DATA_BLOCK "BM_GRW_REC_BOOL"   // DB701
{ S7_Optimized_Access := 'FALSE' }
VERSION : 0.0
// --------------------------------------------------------------------------------
// program:             GRW_REC_BOOL
// description :        bool data for growth record
// name:                mb
// date        :        27.11.09 
// --------------------------------------------------------------------------------
   VAR
      phase_restart : Bool;   // Phase wurde neu gestartet
      phase_spare_02 : Bool;
      phase_spare_03 : Bool;
      phase_spare_04 : Bool;
      phase_spare_05 : Bool;
      phase_spare_06 : Bool;
      phase_spare_07 : Bool;
      phase_spare_08 : Bool;
      phase_spare_09 : Bool;
      phase_spare_10 : Bool;   // pump down
      pd_min_prs_reached : Bool;   // min. Druck erreicht
      pd_failed : Bool;   // Leckrate (0=ok/1=nicht ok)
      pd_new_seed : Bool;   // neuer Impfling bei Prozesstart
      pd_spare_04 : Bool;
      pd_spare_05 : Bool;
      pd_spare_06 : Bool;
      pd_spare_07 : Bool;
      pd_spare_08 : Bool;
      pd_spare_09 : Bool;
      pd_spare_10 : Bool;   // melting
      me_completed : Bool;   // Einschmelzen beendet (von Kamera erkannt)
      me_spare_02 : Bool;
      me_spare_03 : Bool;
      me_spare_04 : Bool;
      me_spare_05 : Bool;
      me_spare_06 : Bool;
      me_spare_07 : Bool;
      me_spare_08 : Bool;
      me_spare_09 : Bool;
      me_spare_10 : Bool;   // dipping
      di_new_seed : Bool;   // alter oder neuer Impfling (0=alt/1=neu)
      di_shield_dn : Bool;   // Trichter ist unten
      di_spare_03 : Bool;
      di_spare_04 : Bool;
      di_spare_05 : Bool;
      di_spare_06 : Bool;
      di_spare_07 : Bool;
      di_spare_08 : Bool;
      di_spare_09 : Bool;
      di_spare_10 : Bool;   // neck
      ne_spare_01 : Bool;
      ne_spare_02 : Bool;
      ne_spare_03 : Bool;
      ne_spare_04 : Bool;
      ne_spare_05 : Bool;
      ne_spare_06 : Bool;
      ne_spare_07 : Bool;
      ne_spare_08 : Bool;
      ne_spare_09 : Bool;
      ne_spare_10 : Bool;   // shoulder
      sh_spare_01 : Bool;
      sh_spare_02 : Bool;
      sh_spare_03 : Bool;
      sh_spare_04 : Bool;
      sh_spare_05 : Bool;
      sh_spare_06 : Bool;
      sh_spare_07 : Bool;
      sh_spare_08 : Bool;
      sh_spare_09 : Bool;
      sh_spare_10 : Bool;   // body
      by_spare_01 : Bool;
      by_spare_02 : Bool;
      by_spare_03 : Bool;
      by_spare_04 : Bool;
      by_spare_05 : Bool;
      by_spare_06 : Bool;
      by_spare_07 : Bool;
      by_spare_08 : Bool;
      by_spare_09 : Bool;
      by_spare_10 : Bool;   // endcone
      ec_spare_01 : Bool;
      ec_spare_02 : Bool;
      ec_spare_03 : Bool;
      ec_spare_04 : Bool;
      ec_spare_05 : Bool;
      ec_spare_06 : Bool;
      ec_spare_07 : Bool;
      ec_spare_08 : Bool;
      ec_spare_09 : Bool;
      ec_spare_10 : Bool;   // shut down
      sd_spare_01 : Bool;
      sd_spare_02 : Bool;
      sd_spare_03 : Bool;
      sd_spare_04 : Bool;
      sd_spare_05 : Bool;
      sd_spare_06 : Bool;
      sd_spare_07 : Bool;
      sd_spare_08 : Bool;
      sd_spare_09 : Bool;
      sd_spare_10 : Bool;   // removal
      re_active : Bool;   // Entnahme wurde ausgef黨rt
      re_spare_02 : Bool;
      re_spare_03 : Bool;
      re_spare_04 : Bool;
      re_spare_05 : Bool;
      re_spare_06 : Bool;
      re_spare_07 : Bool;
      re_spare_08 : Bool;
      re_spare_09 : Bool;
      re_spare_10 : Bool;   // melting back
      mb_spare_01 : Bool;
      mb_spare_02 : Bool;
      mb_spare_03 : Bool;
      mb_spare_04 : Bool;
      mb_spare_05 : Bool;
      mb_spare_06 : Bool;
      mb_spare_07 : Bool;
      mb_spare_08 : Bool;
      mb_spare_09 : Bool;
      mb_spare_10 : Bool;   // interne Speicherbits
      pd_sps_spare_01 : Bool;
      pd_sps_spare_02 : Bool;
      pd_sps_spare_03 : Bool;
      pd_sps_spare_04 : Bool;
      pd_sps_spare_05 : Bool;
      pd_sps_spare_06 : Bool;
      pd_sps_spare_07 : Bool;
      pd_sps_spare_08 : Bool;
      pd_sps_spare_09 : Bool;
      pd_sps_spare_10 : Bool;
      me_sps_spare_01 : Bool;
      me_sps_spare_02 : Bool;
      me_sps_spare_03 : Bool;
      me_sps_spare_04 : Bool;
      me_sps_spare_05 : Bool;
      me_sps_spare_06 : Bool;
      me_sps_spare_07 : Bool;
      me_sps_spare_08 : Bool;
      me_sps_spare_09 : Bool;
      me_sps_spare_10 : Bool;
      di_init_melt_temp : Bool;   // speichern Anfangs-Schmelzbadtemp. ausgef黨rt
      di_time_until_dip : Bool;   // speichern der Zeit bis Impfling in Schmelze ausgef黨rt
      di_sps_spare_03 : Bool;
      di_sps_spare_04 : Bool;
      di_sps_spare_05 : Bool;
      di_sps_spare_06 : Bool;
      di_sps_spare_07 : Bool;
      di_sps_spare_08 : Bool;
      di_sps_spare_09 : Bool;
      di_sps_spare_10 : Bool;
      ne_init_xt_pos : Bool;   // speichern Anfangs-Kristallpos. ausgef黨rt
      ne_init_cr_pos : Bool;   // speichern Anfangs-Tiegelposition ausgef黨rt
      ne_init_melt_temp : Bool;   // speichern Anfangs-Schmelzbadtemp. ausgef黨rt
      ne_low_temp_inc : Bool;   // speichern niedrigstes Temp.Inkrement ausgef黨rt
      ne_init_htr_temp : Bool;   // speichern Heizertemp
      ne_sps_spare_06 : Bool;
      ne_sps_spare_07 : Bool;
      ne_sps_spare_08 : Bool;
      ne_sps_spare_09 : Bool;
      ne_sps_spare_10 : Bool;
      sh_start_dia : Bool;   // speichern Startdurchmesser ausgef黨rt
      sh_init_htr_temp : Bool;   // speichern Heizertemp
      sh_sps_spare_03 : Bool;
      sh_sps_spare_04 : Bool;
      sh_sps_spare_05 : Bool;
      sh_sps_spare_06 : Bool;
      sh_sps_spare_07 : Bool;
      sh_sps_spare_08 : Bool;
      sh_sps_spare_09 : Bool;
      sh_sps_spare_10 : Bool;
      by_low_temp_inc : Bool;   // speichern niedrigstes Temp.Inkrement ausgef黨rt
      by_first_dia : Bool;   // speichern Startdurchmesser ausgef黨rt
      by_init_htr_temp : Bool;   // speichern Heizertemp
      by_sps_spare_04 : Bool;
      by_sps_spare_05 : Bool;
      by_sps_spare_06 : Bool;
      by_sps_spare_07 : Bool;
      by_sps_spare_08 : Bool;
      by_sps_spare_09 : Bool;
      by_sps_spare_10 : Bool;
      ec_init_htr_temp : Bool;   // speichern Heizertemp
      ec_sps_spare_02 : Bool;
      ec_sps_spare_03 : Bool;
      ec_sps_spare_04 : Bool;
      ec_sps_spare_05 : Bool;
      ec_sps_spare_06 : Bool;
      ec_sps_spare_07 : Bool;
      ec_sps_spare_08 : Bool;
      ec_sps_spare_09 : Bool;
      ec_sps_spare_10 : Bool;
      sd_sps_spare_01 : Bool;
      sd_sps_spare_02 : Bool;
      sd_sps_spare_03 : Bool;
      sd_sps_spare_04 : Bool;
      sd_sps_spare_05 : Bool;
      sd_sps_spare_06 : Bool;
      sd_sps_spare_07 : Bool;
      sd_sps_spare_08 : Bool;
      sd_sps_spare_09 : Bool;
      sd_sps_spare_10 : Bool;
      re_next_cr_pos : Bool;   // speichern Tiegelposition f黵 n鋍hstes Ankeimen ausgef黨rt
      re_sps_spare_02 : Bool;
      re_sps_spare_03 : Bool;
      re_sps_spare_04 : Bool;
      re_sps_spare_05 : Bool;
      re_sps_spare_06 : Bool;
      re_sps_spare_07 : Bool;
      re_sps_spare_08 : Bool;
      re_sps_spare_09 : Bool;
      re_sps_spare_10 : Bool;
      mb_sps_spare_01 : Bool;
      mb_sps_spare_02 : Bool;
      mb_sps_spare_03 : Bool;
      mb_sps_spare_04 : Bool;
      mb_sps_spare_05 : Bool;
      mb_sps_spare_06 : Bool;
      mb_sps_spare_07 : Bool;
      mb_sps_spare_08 : Bool;
      mb_sps_spare_09 : Bool;
      mb_sps_spare_10 : Bool;
   END_VAR
BEGIN
END_DATA_BLOCK

DATA_BLOCK "BM_GRW_REC_DINT"   // DB702
{ S7_Optimized_Access := 'FALSE' }
VERSION : 0.0
// --------------------------------------------------------------------------------
// program     :        GRW_REC_DINT
// description :        dint data for growth record
// name        :        mb
// date        :        27.11.09
// --------------------------------------------------------------------------------
   VAR
      elapsed_time : DInt;   // gesamte Prozesszeit
      phase_spare_02 : DInt;
      phase_spare_03 : DInt;
      phase_spare_04 : DInt;
      phase_spare_05 : DInt;
      phase_spare_06 : DInt;
      phase_spare_07 : DInt;
      phase_spare_08 : DInt;
      phase_spare_09 : DInt;
      phase_spare_10 : DInt;
      pd_elapsed_time : DInt;   // insgesamt vergangene Prozesszeit
      pd_phase_time : DInt;   // aktuelle/letzte Phasendauer
      pd_to_min_prs : DInt;   // Zeit bis Enddruck erreicht
      pd_retry : DInt;
      pd_spare_05 : DInt;
      pd_spare_06 : DInt;
      pd_spare_07 : DInt;
      pd_spare_08 : DInt;
      pd_spare_09 : DInt;
      pd_spare_10 : DInt;
      me_elapsed_time : DInt;   // insgesamt vergangene Prozesszeit
      me_phase_time : DInt;   // aktuelle/letzte Phasendauer
      me_melt_time : DInt;   // Zeit bis Aufschmelzen beendet
      me_spare_04 : DInt;
      me_spare_05 : DInt;
      me_spare_06 : DInt;
      me_spare_07 : DInt;
      me_spare_08 : DInt;
      me_spare_09 : DInt;
      me_spare_10 : DInt;
      di_elapsed_time : DInt;   // insgesamt vergangene Prozesszeit
      di_phase_time : DInt;   // aktuelle/letzte Phasendauer
      di_shield_dn : DInt;   // Zeit bis Trichter unten
      di_time_until_dip : DInt;   // Zeit bis Impfling in Schmelze
      di_spare_05 : DInt;
      di_spare_06 : DInt;
      di_spare_07 : DInt;
      di_spare_08 : DInt;
      di_spare_09 : DInt;
      di_spare_10 : DInt;
      ne_elapsed_time : DInt;   // insgesamt vergangene Prozesszeit
      ne_phase_time : DInt;   // aktuelle/letzte Phasendauer
      ne_spare_03 : DInt;
      ne_spare_04 : DInt;
      ne_spare_05 : DInt;
      ne_spare_06 : DInt;
      ne_spare_07 : DInt;
      ne_spare_08 : DInt;
      ne_spare_09 : DInt;
      ne_spare_10 : DInt;
      sh_elapsed_time : DInt;   // insgesamt vergangene Prozesszeit
      sh_phase_time : DInt;   // aktuelle/letzte Phasendauer
      sh_spare_03 : DInt;
      sh_spare_04 : DInt;
      sh_spare_05 : DInt;
      sh_spare_06 : DInt;
      sh_spare_07 : DInt;
      sh_spare_08 : DInt;
      sh_spare_09 : DInt;
      sh_spare_10 : DInt;
      by_elapsed_time : DInt;   // insgesamt vergangene Prozesszeit
      by_phase_time : DInt;   // aktuelle/letzte Phasendauer
      by_spare_03 : DInt;
      by_spare_04 : DInt;
      by_spare_05 : DInt;
      by_spare_06 : DInt;
      by_spare_07 : DInt;
      by_spare_08 : DInt;
      by_spare_09 : DInt;
      by_spare_10 : DInt;
      ec_elapsed_time : DInt;   // insgesamt vergangene Prozesszeit
      ec_phase_time : DInt;   // aktuelle/letzte Phasendauer
      ec_spare_03 : DInt;
      ec_spare_04 : DInt;
      ec_spare_05 : DInt;
      ec_spare_06 : DInt;
      ec_spare_07 : DInt;
      ec_spare_08 : DInt;
      ec_spare_09 : DInt;
      ec_spare_10 : DInt;
      sd_elapsed_time : DInt;   // insgesamt vergangene Prozesszeit
      sd_phase_time : DInt;   // aktuelle/letzte Phasendauer
      sd_spare_03 : DInt;
      sd_spare_04 : DInt;
      sd_spare_05 : DInt;
      sd_spare_06 : DInt;
      sd_spare_07 : DInt;
      sd_spare_08 : DInt;
      sd_spare_09 : DInt;
      sd_spare_10 : DInt;
      re_elapsed_time : DInt;   // insgesamt vergangene Prozesszeit
      re_phase_time : DInt;   // aktuelle/letzte Phasendauer
      re_spare_03 : DInt;
      re_spare_04 : DInt;
      re_spare_05 : DInt;
      re_spare_06 : DInt;
      re_spare_07 : DInt;
      re_spare_08 : DInt;
      re_spare_09 : DInt;
      re_spare_10 : DInt;
      mb_elapsed_time : DInt;   // insgesamt vergangene Prozesszeit
      mb_phase_time : DInt;   // aktuelle/letzte Phasendauer
      mb_spare_03 : DInt;
      mb_spare_04 : DInt;
      mb_spare_05 : DInt;
      mb_spare_06 : DInt;
      mb_spare_07 : DInt;
      mb_spare_08 : DInt;
      mb_spare_09 : DInt;
      mb_spare_10 : DInt;
   END_VAR
BEGIN
END_DATA_BLOCK

DATA_BLOCK "BM_GRW_REC_REAL"   // DB703
{ S7_Optimized_Access := 'FALSE' }
VERSION : 0.0
// --------------------------------------------------------------------------------
// program:             GRW_REC_REAL
// description :        REAL data for growth record
// name:                mb
// date        :        23.11.09
// --------------------------------------------------------------------------------
   VAR
      htr_pwr_csp : Real;   // heater power consumption
      ar_gas_csp : Real;   // argon gas consumption
      phase_spare_03 : Real;
      phase_spare_04 : Real;
      phase_spare_05 : Real;
      phase_spare_06 : Real;
      phase_spare_07 : Real;
      phase_spare_08 : Real;
      phase_spare_09 : Real;
      phase_spare_10 : Real;
      phase_spare_11 : Real;
      phase_spare_12 : Real;
      phase_spare_13 : Real;
      phase_spare_14 : Real;
      phase_spare_15 : Real;
      phase_spare_16 : Real;
      phase_spare_17 : Real;
      phase_spare_18 : Real;
      phase_spare_19 : Real;
      phase_spare_20 : Real;
      phase_spare_21 : Real;
      phase_spare_22 : Real;
      phase_spare_23 : Real;
      phase_spare_24 : Real;
      phase_spare_25 : Real;
      phase_spare_26 : Real;
      phase_spare_27 : Real;
      phase_spare_28 : Real;
      phase_spare_29 : Real;
      phase_spare_30 : Real;
      phase_spare_31 : Real;
      phase_spare_32 : Real;
      phase_spare_33 : Real;
      phase_spare_34 : Real;
      phase_spare_35 : Real;
      phase_spare_36 : Real;
      phase_spare_37 : Real;
      phase_spare_38 : Real;
      phase_spare_39 : Real;
      phase_spare_40 : Real;
      pd_final_prs : Real;   // erreichter Enddruck
      pd_leakrate : Real;   // Leckrate
      pd_spare_03 : Real;
      pd_spare_04 : Real;
      pd_spare_05 : Real;
      pd_spare_06 : Real;
      pd_spare_07 : Real;
      pd_spare_08 : Real;
      pd_spare_09 : Real;
      pd_spare_10 : Real;
      pd_spare_11 : Real;
      pd_spare_12 : Real;
      pd_spare_13 : Real;
      pd_spare_14 : Real;
      pd_spare_15 : Real;
      pd_spare_16 : Real;
      pd_spare_17 : Real;
      pd_spare_18 : Real;
      pd_spare_19 : Real;
      pd_spare_20 : Real;
      pd_spare_21 : Real;
      pd_spare_22 : Real;
      pd_spare_23 : Real;
      pd_spare_24 : Real;
      pd_spare_25 : Real;
      pd_spare_26 : Real;
      pd_spare_27 : Real;
      pd_spare_28 : Real;
      pd_spare_29 : Real;
      pd_spare_30 : Real;
      pd_spare_31 : Real;
      pd_spare_32 : Real;
      pd_spare_33 : Real;
      pd_spare_34 : Real;
      pd_spare_35 : Real;
      pd_spare_36 : Real;
      pd_spare_37 : Real;
      pd_spare_38 : Real;
      pd_spare_39 : Real;
      pd_spare_40 : Real;
      me_spare_01 : Real;
      me_spare_02 : Real;
      me_spare_03 : Real;
      me_spare_04 : Real;
      me_spare_05 : Real;
      me_spare_06 : Real;
      me_spare_07 : Real;
      me_spare_08 : Real;
      me_spare_09 : Real;
      me_spare_10 : Real;
      me_spare_11 : Real;
      me_spare_12 : Real;
      me_spare_13 : Real;
      me_spare_14 : Real;
      me_spare_15 : Real;
      me_spare_16 : Real;
      me_spare_17 : Real;
      me_spare_18 : Real;
      me_spare_19 : Real;
      me_spare_20 : Real;
      me_spare_21 : Real;
      me_spare_22 : Real;
      me_spare_23 : Real;
      me_spare_24 : Real;
      me_spare_25 : Real;
      me_spare_26 : Real;
      me_spare_27 : Real;
      me_spare_28 : Real;
      me_spare_29 : Real;
      me_spare_30 : Real;
      me_spare_31 : Real;
      me_spare_32 : Real;
      me_spare_33 : Real;
      me_spare_34 : Real;
      me_spare_35 : Real;
      me_spare_36 : Real;
      me_spare_37 : Real;
      me_spare_38 : Real;
      me_spare_39 : Real;
      me_spare_40 : Real;
      di_init_melt_temp : Real;   // Anfangs-Schmelzbadtemp.
      di_final_htr_1_pwr : Real;   // Heizer 1 Leistung am Phasenende
      di_spare_03 : Real;
      di_spare_04 : Real;
      di_spare_05 : Real;
      di_spare_06 : Real;
      di_spare_07 : Real;
      di_spare_08 : Real;
      di_spare_09 : Real;
      di_spare_10 : Real;
      di_spare_11 : Real;
      di_spare_12 : Real;
      di_spare_13 : Real;
      di_spare_14 : Real;
      di_spare_15 : Real;
      di_spare_16 : Real;
      di_spare_17 : Real;
      di_spare_18 : Real;
      di_spare_19 : Real;
      di_spare_20 : Real;
      di_spare_21 : Real;
      di_spare_22 : Real;
      di_spare_23 : Real;
      di_spare_24 : Real;
      di_spare_25 : Real;
      di_spare_26 : Real;
      di_spare_27 : Real;
      di_spare_28 : Real;
      di_spare_29 : Real;
      di_spare_30 : Real;
      di_spare_31 : Real;
      di_spare_32 : Real;
      di_spare_33 : Real;
      di_spare_34 : Real;
      di_spare_35 : Real;
      di_spare_36 : Real;
      di_spare_37 : Real;
      di_spare_38 : Real;
      di_spare_39 : Real;
      di_spare_40 : Real;
      ne_init_cr_pos : Real;   // Anfangs-Tiegelpos.
      ne_init_melt_temp : Real;   // Anfangs-Schmelzbadtemp.
      ne_final_melt_temp : Real;   // finale-Schmelzbadtemp.
      ne_low_temp_inc : Real;   // niedrigstes Temp.Inc.
      ne_final_temp_inc : Real;   // finales Temp.Inc.
      ne_phase_avg_spd : Real;   // Durchschnittl. Ziehgeschwindigkeit (gesamte Halsl鋘ge)
      ne_final_avg_spd : Real;   // finale Durchschnittl. Ziehgeschwindigkeit
      ne_final_htr_1_pwr : Real;   // Heizer 1 Leistung am Phasenende
      ne_spare_09 : Real;
      ne_spare_10 : Real;
      ne_spare_11 : Real;
      ne_spare_12 : Real;
      ne_spare_13 : Real;
      ne_spare_14 : Real;
      ne_spare_15 : Real;
      ne_spare_16 : Real;
      ne_spare_17 : Real;
      ne_spare_18 : Real;
      ne_spare_19 : Real;
      ne_spare_20 : Real;
      ne_spare_21 : Real;
      ne_spare_22 : Real;
      ne_spare_23 : Real;
      ne_spare_24 : Real;
      ne_spare_25 : Real;
      ne_spare_26 : Real;
      ne_spare_27 : Real;
      ne_spare_28 : Real;
      ne_spare_29 : Real;
      ne_spare_30 : Real;
      ne_spare_31 : Real;
      ne_spare_32 : Real;
      ne_spare_33 : Real;
      ne_spare_34 : Real;
      ne_spare_35 : Real;
      ne_spare_36 : Real;
      ne_spare_37 : Real;
      ne_spare_38 : Real;
      ne_spare_39 : Real;
      ne_spare_40 : Real;
      sh_phase_avg_grth : Real;   // Durchschnittl. Wachstumsgeschwindigkeit (gesamte Schulter)
      sh_final_temp_inc : Real;   // finales Temp.Inc.
      sh_weight : Real;   // Gewicht der Schulter
      sh_final_htr_1_pwr : Real;   // Heizer 1 Leistung am Phasenende
      sh_spare_05 : Real;
      sh_spare_06 : Real;
      sh_spare_07 : Real;
      sh_spare_08 : Real;
      sh_spare_09 : Real;
      sh_spare_10 : Real;
      sh_spare_11 : Real;
      sh_spare_12 : Real;
      sh_spare_13 : Real;
      sh_spare_14 : Real;
      sh_spare_15 : Real;
      sh_spare_16 : Real;
      sh_spare_17 : Real;
      sh_spare_18 : Real;
      sh_spare_19 : Real;
      sh_spare_20 : Real;
      sh_spare_21 : Real;
      sh_spare_22 : Real;
      sh_spare_23 : Real;
      sh_spare_24 : Real;
      sh_spare_25 : Real;
      sh_spare_26 : Real;
      sh_spare_27 : Real;
      sh_spare_28 : Real;
      sh_spare_29 : Real;
      sh_spare_30 : Real;
      sh_spare_31 : Real;
      sh_spare_32 : Real;
      sh_spare_33 : Real;
      sh_spare_34 : Real;
      sh_spare_35 : Real;
      sh_spare_36 : Real;
      sh_spare_37 : Real;
      sh_spare_38 : Real;
      sh_spare_39 : Real;
      sh_spare_40 : Real;
      by_phase_avg_spd : Real;   // Durchschnittl. Ziehgeschwindigkeit (gesamt)
      by_final_avg_spd : Real;   // finale Durchschnittl. Ziehgeschwindigkeit
      by_low_temp_inc : Real;   // niedrigstes Temp.Inc.
      by_final_temp_inc : Real;   // finales Temp.Inc.
      by_avg_dia : Real;   // Durchschnittl. Durchmesser
      by_weight : Real;   // Gewicht vom Stab
      by_lenght : Real;   // Stabl鋘ge
      by_total_length : Real;   // Gesamtl鋘ge
      by_rem_cr_wgt : Real;   // verbleibende Siliziummenge im Tiegel
      by_final_cr_pos : Real;   // finale Tiegelpos.
      by_final_htr_1_pwr : Real;   // Heizer 1 Leistung am Phasenende
      by_spare_12 : Real;
      by_spare_13 : Real;
      by_spare_14 : Real;
      by_spare_15 : Real;
      by_spare_16 : Real;
      by_spare_17 : Real;
      by_spare_18 : Real;
      by_spare_19 : Real;
      by_spare_20 : Real;
      by_spare_21 : Real;
      by_spare_22 : Real;
      by_spare_23 : Real;
      by_spare_24 : Real;
      by_spare_25 : Real;
      by_spare_26 : Real;
      by_spare_27 : Real;
      by_spare_28 : Real;
      by_spare_29 : Real;
      by_spare_30 : Real;
      by_spare_31 : Real;
      by_spare_32 : Real;
      by_spare_33 : Real;
      by_spare_34 : Real;
      by_spare_35 : Real;
      by_spare_36 : Real;
      by_spare_37 : Real;
      by_spare_38 : Real;
      by_spare_39 : Real;
      by_spare_40 : Real;
      ec_phase_avg_spd : Real;   // Durchschnittl. Ziehgeschwindigkeit (gesamt)
      ec_final_temp_inc : Real;   // finales Temp.Inc.
      ec_weight : Real;   // Gewicht vom Endkonus
      ec_rem_cr_wgt : Real;   // verbleibende Siliziummenge im Tiegel
      ec_final_htr_1_pwr : Real;   // Heizer 1 Leistung am Phasenende
      ec_spare_06 : Real;
      ec_spare_07 : Real;
      ec_spare_08 : Real;
      ec_spare_09 : Real;
      ec_spare_10 : Real;
      ec_spare_11 : Real;
      ec_spare_12 : Real;
      ec_spare_13 : Real;
      ec_spare_14 : Real;
      ec_spare_15 : Real;
      ec_spare_16 : Real;
      ec_spare_17 : Real;
      ec_spare_18 : Real;
      ec_spare_19 : Real;
      ec_spare_20 : Real;
      ec_spare_21 : Real;
      ec_spare_22 : Real;
      ec_spare_23 : Real;
      ec_spare_24 : Real;
      ec_spare_25 : Real;
      ec_spare_26 : Real;
      ec_spare_27 : Real;
      ec_spare_28 : Real;
      ec_spare_29 : Real;
      ec_spare_30 : Real;
      ec_spare_31 : Real;
      ec_spare_32 : Real;
      ec_spare_33 : Real;
      ec_spare_34 : Real;
      ec_spare_35 : Real;
      ec_spare_36 : Real;
      ec_spare_37 : Real;
      ec_spare_38 : Real;
      ec_spare_39 : Real;
      ec_spare_40 : Real;
      sd_spare_01 : Real;
      sd_spare_02 : Real;
      sd_spare_03 : Real;
      sd_spare_04 : Real;
      sd_spare_05 : Real;
      sd_spare_06 : Real;
      sd_spare_07 : Real;
      sd_spare_08 : Real;
      sd_spare_09 : Real;
      sd_spare_10 : Real;
      sd_spare_11 : Real;
      sd_spare_12 : Real;
      sd_spare_13 : Real;
      sd_spare_14 : Real;
      sd_spare_15 : Real;
      sd_spare_16 : Real;
      sd_spare_17 : Real;
      sd_spare_18 : Real;
      sd_spare_19 : Real;
      sd_spare_20 : Real;
      sd_spare_21 : Real;
      sd_spare_22 : Real;
      sd_spare_23 : Real;
      sd_spare_24 : Real;
      sd_spare_25 : Real;
      sd_spare_26 : Real;
      sd_spare_27 : Real;
      sd_spare_28 : Real;
      sd_spare_29 : Real;
      sd_spare_30 : Real;
      sd_spare_31 : Real;
      sd_spare_32 : Real;
      sd_spare_33 : Real;
      sd_spare_34 : Real;
      sd_spare_35 : Real;
      sd_spare_36 : Real;
      sd_spare_37 : Real;
      sd_spare_38 : Real;
      sd_spare_39 : Real;
      sd_spare_40 : Real;
      re_next_cr_pos : Real;   // n鋍hste Tiegelpos.
      re_final_htr_1_pwr : Real;   // Heizer 1 Leistung am Phasenende
      re_spare_03 : Real;
      re_spare_04 : Real;
      re_spare_05 : Real;
      re_spare_06 : Real;
      re_spare_07 : Real;
      re_spare_08 : Real;
      re_spare_09 : Real;
      re_spare_10 : Real;
      re_spare_11 : Real;
      re_spare_12 : Real;
      re_spare_13 : Real;
      re_spare_14 : Real;
      re_spare_15 : Real;
      re_spare_16 : Real;
      re_spare_17 : Real;
      re_spare_18 : Real;
      re_spare_19 : Real;
      re_spare_20 : Real;
      re_spare_21 : Real;
      re_spare_22 : Real;
      re_spare_23 : Real;
      re_spare_24 : Real;
      re_spare_25 : Real;
      re_spare_26 : Real;
      re_spare_27 : Real;
      re_spare_28 : Real;
      re_spare_29 : Real;
      re_spare_30 : Real;
      re_spare_31 : Real;
      re_spare_32 : Real;
      re_spare_33 : Real;
      re_spare_34 : Real;
      re_spare_35 : Real;
      re_spare_36 : Real;
      re_spare_37 : Real;
      re_spare_38 : Real;
      re_spare_39 : Real;
      re_spare_40 : Real;
      mb_phase_avg_spd : Real;
      mb_final_cr_pos : Real;
      mb_spare_03 : Real;
      mb_spare_04 : Real;
      mb_spare_05 : Real;
      mb_spare_06 : Real;
      mb_spare_07 : Real;
      mb_spare_08 : Real;
      mb_spare_09 : Real;
      mb_spare_10 : Real;
      mb_spare_11 : Real;
      mb_spare_12 : Real;
      mb_spare_13 : Real;
      mb_spare_14 : Real;
      mb_spare_15 : Real;
      mb_spare_16 : Real;
      mb_spare_17 : Real;
      mb_spare_18 : Real;
      mb_spare_19 : Real;
      mb_spare_20 : Real;
      mb_spare_21 : Real;
      mb_spare_22 : Real;
      mb_spare_23 : Real;
      mb_spare_24 : Real;
      mb_spare_25 : Real;
      mb_spare_26 : Real;
      mb_spare_27 : Real;
      mb_spare_28 : Real;
      mb_spare_29 : Real;
      mb_spare_30 : Real;
      mb_spare_31 : Real;
      mb_spare_32 : Real;
      mb_spare_33 : Real;
      mb_spare_34 : Real;
      mb_spare_35 : Real;
      mb_spare_36 : Real;
      mb_spare_37 : Real;
      mb_spare_38 : Real;
      mb_spare_39 : Real;
      mb_spare_40 : Real;   // interne Speicherwerte
      pd_sps_spare_01 : Real;
      pd_sps_spare_02 : Real;
      pd_sps_spare_03 : Real;
      pd_sps_spare_04 : Real;
      pd_sps_spare_05 : Real;
      pd_sps_spare_06 : Real;
      pd_sps_spare_07 : Real;
      pd_sps_spare_08 : Real;
      pd_sps_spare_09 : Real;
      pd_sps_spare_10 : Real;
      me_sps_spare_01 : Real;
      me_sps_spare_02 : Real;
      me_sps_spare_03 : Real;
      me_sps_spare_04 : Real;
      me_sps_spare_05 : Real;
      me_sps_spare_06 : Real;
      me_sps_spare_07 : Real;
      me_sps_spare_08 : Real;
      me_sps_spare_09 : Real;
      me_sps_spare_10 : Real;
      di_sps_spare_01 : Real;
      di_sps_spare_02 : Real;
      di_sps_spare_03 : Real;
      di_sps_spare_04 : Real;
      di_sps_spare_05 : Real;
      di_sps_spare_06 : Real;
      di_sps_spare_07 : Real;
      di_sps_spare_08 : Real;
      di_sps_spare_09 : Real;
      di_sps_spare_10 : Real;
      ne_sps_init_xt_pos : Real;   // Anfangs-Kristallpos.
      ne_sps_init_htr_temp : Real;   // Anfangs-Heizertemp
      ne_sps_spare_03 : Real;
      ne_sps_spare_04 : Real;
      ne_sps_spare_05 : Real;
      ne_sps_spare_06 : Real;
      ne_sps_spare_07 : Real;
      ne_sps_spare_08 : Real;
      ne_sps_spare_09 : Real;
      ne_sps_spare_10 : Real;
      sh_sps_start_dia : Real;   // Startdurchnesser (nur Speicher f黵 Berechnung)
      sh_sps_init_htr_temp : Real;   // Anfangs-Heizertemp
      sh_sps_spare_03 : Real;
      sh_sps_spare_04 : Real;
      sh_sps_spare_05 : Real;
      sh_sps_spare_06 : Real;
      sh_sps_spare_07 : Real;
      sh_sps_spare_08 : Real;
      sh_sps_spare_09 : Real;
      sh_sps_spare_10 : Real;
      by_first_dia : Real;   // Startdurchmesser (nur Speicher f黵 Berechnung)
      by_start_wgt : Real;   // Startgewicht (nur Speicher f黵 Berechnung)
      by_sps_init_htr_temp : Real;   // Anfangs-Heizertemp
      by_sps_spare_04 : Real;
      by_sps_spare_05 : Real;
      by_sps_spare_06 : Real;
      by_sps_spare_07 : Real;
      by_sps_spare_08 : Real;
      by_sps_spare_09 : Real;
      by_sps_spare_10 : Real;
      ec_sps_init_htr_temp : Real;   // Anfangs-Heizertemp
      ec_sps_spare_02 : Real;
      ec_sps_spare_03 : Real;
      ec_sps_spare_04 : Real;
      ec_sps_spare_05 : Real;
      ec_sps_spare_06 : Real;
      ec_sps_spare_07 : Real;
      ec_sps_spare_08 : Real;
      ec_sps_spare_09 : Real;
      ec_sps_spare_10 : Real;
      sd_sps_spare_01 : Real;
      sd_sps_spare_02 : Real;
      sd_sps_spare_03 : Real;
      sd_sps_spare_04 : Real;
      sd_sps_spare_05 : Real;
      sd_sps_spare_06 : Real;
      sd_sps_spare_07 : Real;
      sd_sps_spare_08 : Real;
      sd_sps_spare_09 : Real;
      sd_sps_spare_10 : Real;
      re_sps_rem_si_wgt : Real;
      re_sps_spare_02 : Real;
      re_sps_spare_03 : Real;
      re_sps_spare_04 : Real;
      re_sps_spare_05 : Real;
      re_sps_spare_06 : Real;
      re_sps_spare_07 : Real;
      re_sps_spare_08 : Real;
      re_sps_spare_09 : Real;
      re_sps_spare_10 : Real;
      mb_sps_spare_01 : Real;
      mb_sps_spare_02 : Real;
      mb_sps_spare_03 : Real;
      mb_sps_spare_04 : Real;
      mb_sps_spare_05 : Real;
      mb_sps_spare_06 : Real;
      mb_sps_spare_07 : Real;
      mb_sps_spare_08 : Real;
      mb_sps_spare_09 : Real;
      mb_sps_spare_10 : Real;
   END_VAR
BEGIN
END_DATA_BLOCK

DATA_BLOCK "IDI"   // DB896
{ S7_Optimized_Access := 'FALSE' }
VERSION : 0.0
// --------------------------------------------------------------------------------
// program:             IDI
// description :        automatically generated IDI
// name:                hp
// date        :        03.02.2021
// 
// revision:
// name:
// date:
//                     (c)CGS
// --------------------------------------------------------------------------------
   VAR
      CB_FLT_DC24V_K2 : Bool;   // HDI def M 72.0: fault circuit breakers DC 24V 1=OK
      CB_FLT_AC400V_K2 : Bool;   // HDI def M 72.1: fault circuit breakers AC 400V 1=OK
      SPARE_16_2 : Bool;   // HDI def M 72.4: spare digital input
      CB_FLT_AC230V : Bool;   // HDI def M 72.3: fault circuit breakers AC 230V 1=OK
      SPARE_16_4 : Bool;   // HDI def M 72.4: spare digital input
      SPARE_16_5 : Bool;   // HDI def M 72.5: spare digital input
      SPARE_16_6 : Bool;   // HDI def M 72.6: spare digital input
      SPARE_16_7 : Bool;   // HDI def M 72.7: spare digital input
      SPARE_17_0 : Bool;   // HDI def M 73.0: spare digital input
      UPS_24V_ALM : Bool;   // HDI def M 73.1: alarm dc-usv
      UPS_24V_NRM : Bool;   // HDI def M 73.2: main line ready buffered dc-usv
      EMO : Bool;   // HDI def M 73.3: Emergency off (1=ok)
      EMS : Bool;   // HDI def M 73.4: Emergency stop handling drives (1=ok)
      SPARE_17_5 : Bool;   // HDI def M 73.5: spare digital input
      SPARE_17_6 : Bool;   // HDI def M 73.6: spare digital input
      SPARE_17_7 : Bool;   // HDI def M 73.7: spare digital input
      P1_WRN : Bool;   // HDI def M 74.0: pump unit (P1) warning
      P1_FLT : Bool;   // HDI def M 74.1: pump unit (P1) error
      P1_IS_ON : Bool;   // HDI def M 74.2: pump unit (P1) running
      P1_WD : Bool;   // HDI def M 74.3: pump unit (P1) watchdog
      FIL_APS : Bool;   // HDI def M 74.4: pressure filter 1000 mbar
      MON_TMP_P2 : Bool;   // HDI def M 74.5: temperature monitoring P2
      MON_TMP_P1 : Bool;   // HDI def M 74.6: temperature monitoring P1
      SPARE_18_7 : Bool;   // HDI def M 74.7: spare digital input
      FCH_LFT_SDL_NUT : Bool;   // HDI def M 88.0: safety limit switch furnace chamber lift spindle nut
      LS_FCH_LFT_DN : Bool;   // HDI def M 88.1: limit switch furnace chamber lift down
      LS_FCH_HOOK_WORK : Bool;   // HDI def M 88.2: limit switch furnace chamber hook in working position
      LS_FCH_HOOK_HOME : Bool;   // HDI def M 88.3: limit switch furnace chamber hook in home position
      LS_TEC_FLG_DN : Bool;   // HDI def M 88.4: limit switch technolgy flange down
      TEC_FLG_SDL_NUT : Bool;   // HDI def M 88.5: safety limit switch technolgy flange lift spindle nut
      LS_V11_COV_OP : Bool;   // HDI def M 88.6: Cover V11 opened (isolation valve feeder)
      LS_V11_COV_CL : Bool;   // HDI def M 88.7: Cover V11 closed (isolation valve feeder)
      GCH_APS : Bool;   // HDI def M 89.0: pressure gate chamber 1000 mbar
      FCH_APS : Bool;   // HDI def M 89.1: pressure furnace chamber 1000 mbar
      FDR_APS : Bool;   // HDI def M 89.2: pressure feeder 1000 mbar
      FIL_2_APS : Bool;   // HDI def M 89.3: atmospheric pressure filter 2
      SPARE_33_4 : Bool;   // HDI def M 89.4: spare
      SPARE_33_5 : Bool;   // HDI def M 89.5: spare
      LS_V2_1_OP : Bool;   // HDI def M 89.6: valve position v2.1 fce chamber
      LS_V2_1_CL : Bool;   // HDI def M 89.7: valve position v2.1 fce chamber
      CB_FLT_AC400V_K5 : Bool;   // HDI def M 90.0: fault circuit breakers AC 400V +K5 1=OK
      CB_FLT_DC24V_K5 : Bool;   // HDI def M 90.1: fault circuit breakers DC 24V +K5 1=OK
      LS_MAG_LFT_UP : Bool;   // HDI def M 90.2: limit switch magnet lift up
      LS_MAG_LFT_DN : Bool;   // HDI def M 90.3: limit switch magnet lift down
      SLS_MAG_LFT : Bool;   // HDI def M 90.4: Safety limit switch magnet lift
      MAG_LFT_SDL_NUT1 : Bool;   // HDI def M 90.5: safety limit switch magnet lift spindle nut 1
      MAG_LFT_SDL_NUT2 : Bool;   // HDI def M 90.6: safety limit switch magnet lift spindle nut 2
      MAG_LFT_SDL_NUT3 : Bool;   // HDI def M 90.7: safety limit switch magnet lift spindle nut 3
      OIL_LVL_CR_SFT : Bool;   // HDI def M 91.0: Crucible shaft min. oil level
      LS_V1_OP : Bool;   // HDI def M 91.1: V1 opened
      LS_V1_CL : Bool;   // HDI def M 91.2: V1 closed
      MP_ENB_K5 : Bool;   // HDI def M 91.3: Mobile panel agree button +K5
      SLS_TEC_FLG_LFT : Bool;   // HDI def M 91.4: Safety limit switch technolgy flange lift
      SLS_FCH_LFT : Bool;   // HDI def M 91.5: Safety limit switch furnace chamber lift
      COMP_AIR_OK : Bool;   // HDI def M 91.6: pressure switch compressed air ok
      COMP_AIR_2_OK : Bool;   // HDI def M 91.7: pressure switch compressed air 2 (ACC) ok
      LS_V1_1_CL : Bool;   // HDI def M 105.0: limit switch valve v1.1 closed
      LS_V1_1_OP : Bool;   // HDI def M 105.1: limit switch valve v1.1 opened
      LS_V3_4_OP : Bool;   // HDI def M 105.2: limit switch valve v3.4 opened
      LS_V3_4_CL : Bool;   // HDI def M 105.3: limit switch valve v3.4 closed
      LS_V3_3_OP : Bool;   // HDI def M 105.4: limit switch valve v3.3 opened
      LS_V3_3_CL : Bool;   // HDI def M 105.5: limit switch valve v3.3 closed
      LS_V2_11_OP : Bool;   // HDI def M 105.6: limit switch valve v2.11 opened
      LS_V2_11_CL : Bool;   // HDI def M 105.7: limit switch valve v2.11 closed
      ACC_FCH_OV_PRS_1 : Bool;   // HDI def M 92.0: ACC furnace overpressure 1
      ACC_FCH_OV_PRS_2 : Bool;   // HDI def M 92.1: ACC furnace overpressure 2
      SPARE_48_2 : Bool;   // HDI def M 92.2: ACC spare
      ACC_WTR_FLW_OUT_OK : Bool;   // HDI def M 92.3: ACC output waterflow ok
      ACC_WTR_FLW_IN_OK : Bool;   // HDI def M 92.4: ACC input waterflow ok
      ACC_WTR_TMP_OUT_OK : Bool;   // HDI def M 92.5: ACC output watertemp. Ok
      OV_PRS_1_FLT : Bool;   // HDI def M 92.6: ACC overpressure 1 error/fault
      OV_PRS_2_FLT : Bool;   // HDI def M 92.7: ACC overpressure 2 error/fault
      ACC_SC_WTR_OK : Bool;   // HDI def M 93.0: ACC safety circuit
      ACC_SC_WTR_ATV : Bool;   // HDI def M 93.1: ACC safety circuit
      ACC_SC_HTR_OK : Bool;   // HDI def M 93.2: ACC safety circuit
      ACC_SC_HTR_ATV : Bool;   // HDI def M 93.3: ACC safety circuit
      ACC_KEY_RST : Bool;   // HDI def M 93.4: ACC reset key
      ACC_CB_FLT_DC24V : Bool;   // HDI def M 93.5: ACC 24V circuit breaker ok
      ACC_UPS_24V_ALM : Bool;   // HDI def M 93.6: ACC UPS OK Normal
      ACC_UPS_24V_NRM : Bool;   // HDI def M 93.7: ACC UPS Alarm
      DPH_RPT_DET_OK : Bool;   // HDI def M 94.0: ACC Diaphraghm rupture detector OK
      ACC_CB_FLT_AC230V : Bool;   // HDI def M 94.1: Fault circuit breakers AC 230V
      SPARE_90_2 : Bool;   // HDI def M 94.2: ACC spare
      SPARE_90_3 : Bool;   // HDI def M 94.3: ACC spare
      SPARE_90_4 : Bool;   // HDI def M 94.4: ACC spare
      SPARE_90_5 : Bool;   // HDI def M 94.5: ACC spare
      SPARE_90_6 : Bool;   // HDI def M 94.6: ACC spare
      SPARE_90_7 : Bool;   // HDI def M 94.7: ACC spare
      FU_P2_RDY : Bool;   // HDI def M 104.0: Frequency converter P2 ready/ no fault
      SPARE_144_1 : Bool;   // HDI def M 104.1: spare digital input
      SPARE_144_2 : Bool;   // HDI def M 104.2: spare digital input
      SPARE_144_3 : Bool;   // HDI def M 104.3: spare digital input
      SPARE_144_4 : Bool;   // HDI def M 104.4: spare digital input
      SPARE_144_5 : Bool;   // HDI def M 104.5: spare digital input
      SPARE_144_6 : Bool;   // HDI def M 104.6: spare digital input
      SPARE_144_7 : Bool;   // HDI def M 104.7: spare digital input
      LS_GCH_UP : Bool;   // HDI def M 95.0: limit switch gate chamber in upper position
      LS_GCH_DN : Bool;   // HDI def M 95.1: limit switch gate chamber in lower position
      LS_GCH_SW_IN : Bool;   // HDI def M 95.2: limit switch gate chamber swivelled in
      LS_GCH_SW_CLN : Bool;   // HDI def M 95.3: limit switch gate chamber swivelled in cleaning pos
      LS_GCH_SW_OUT : Bool;   // HDI def M 95.4: limit switch gate chamber swivelled out
      LS_GCH_SW_LOCK : Bool;   // HDI def M 95.5: limit switch gate chamber swivel locked
      SLS_GCH_LFT : Bool;   // HDI def M 95.6: Safety limit switch gate chamber lift
      LS_TCH_UP : Bool;   // HDI def M 95.7: limit switch top chamber in upper position
      LS_TCH_DN : Bool;   // HDI def M 96.0: limit switch top chamber in lower position
      LS_TCH_SW_IN : Bool;   // HDI def M 96.1: limit switch top chamber swivelled in
      LS_TCH_SW_CLN : Bool;   // HDI def M 96.2: limit switch top chamber swivelled in cleaning pos
      LS_TCH_SW_OUT : Bool;   // HDI def M 96.3: limit switch top chamber swivelled out
      LS_TCH_SW_LOCK : Bool;   // HDI def M 96.4: limit switch top chamber swivel locked
      LS_TCH_TILT_0 : Bool;   // HDI def M 96.5: limit switch top chamber tilt 0?horizental
      LS_TCH_TILT_30 : Bool;   // HDI def M 96.6: limit switch top chamber tilt 30?Cleaning position
      KEY_XT_LFT_SRV : Bool;   // HDI def M 96.7: Key switch service mode crystal lift
      LS_V7_UP : Bool;   // HDI def M 97.0: limit switch gate valve V7 in upper position
      LS_V7_DN : Bool;   // HDI def M 97.1: limit switch gate valve V7 in lower position
      LS_V7_SW_IN : Bool;   // HDI def M 97.2: limit switch gate valve V7 swiveled in
      LS_V7_SW_OUT : Bool;   // HDI def M 97.3: limit switch gate valve V7 swiveled out
      LS_V7_FLP_OP : Bool;   // HDI def M 97.4: limit switch gate valve V7 flap open
      LS_V7_CLN_POS : Bool;   // HDI def M 97.5: limit switch gate valve V7 in cleaning position
      LS_GCH_BEL_UP : Bool;   // HDI def M 97.6: limit switch gate chamber bellow in upper position
      LS_GCH_BEL_DN : Bool;   // HDI def M 97.7: limit switch gate chamber bellow in lower position
      LS_XT_SLID_BW : Bool;   // HDI def M 98.0: limit switch crystal handling slider in home position
      LS_XT_SLID_FW : Bool;   // HDI def M 98.1: limit switch crystal handling slider in work position
      LS_XT_SLID_MID : Bool;   // HDI def M 98.2: limit switch crystal handling slider in middle position
      LS_XT_CLP_CON : Bool;   // HDI def M 98.3: limit switch crystal handling clamps connected
      LS_XT_TILT_90 : Bool;   // HDI def M 98.4: limit switch crystal handling tilt in 90?
      LS_XT_TILT_75 : Bool;   // HDI def M 98.5: limit switch crystal handling tilt in 75?
      LS_UP_XT_CLP_FLT : Bool;   // HDI def M 98.6: limit switch upper crystal clamp fault
      SPARE_275_7 : Bool;   // HDI def M 98.7: spare digital input
      LS_UP_XT_CLP_OP : Bool;   // HDI def M 99.0: limit switch upper crystal clamp open
      LS_UP_XT_CLP_CL : Bool;   // HDI def M 99.1: limit switch upper crystal clamp closed
      LS_UP_XT_CLP_SAVE : Bool;   // HDI def M 99.2: limit switch upper crystal clamp save
      LS_UP_XT_CLP_PLATE : Bool;   // HDI def M 99.3: limit switch upper crystal clamp plate
      LS_LO_XT_CLP_FLT : Bool;   // HDI def M 99.4: limit switch lower crystal clamp fault
      LS_LO_XT_CLP_OP : Bool;   // HDI def M 99.5: limit switch lower crystal clamp open
      LS_LO_XT_CLP_CL : Bool;   // HDI def M 99.6: limit switch lower crystal clamp closed
      LS_LO_XT_CLP_SAVE : Bool;   // HDI def M 99.7: limit switch lower crystal clamp save
      LS_LO_XT_CLP_PLATE : Bool;   // HDI def M 100.0: limit switch upper crystal clamp plate
      LS_HOI_TOOL_INST : Bool;   // HDI def M 100.1: limit switch HOI tool installed
      XT_DRP_OUT_PRT_1_CL : Bool;   // HDI def M 100.2: crystal drop out protection 1 closed (upper left side)
      XT_DRP_OUT_PRT_1_OP : Bool;   // HDI def M 100.3: crystal drop out protection 1 opened (upper left side)
      XT_DRP_OUT_PRT_2_CL : Bool;   // HDI def M 100.4: crystal drop out protection 2 closed (upper right side)
      XT_DRP_OUT_PRT_2_OP : Bool;   // HDI def M 100.5: crystal drop out protection 2 opened (upper right side)
      CB_FLT_AC400V_K8 : Bool;   // HDI def M 100.6: fault circuit breakers AC 400V 1=OK
      CB_FLT_DC24V_K8 : Bool;   // HDI def M 100.7: fault circuit breakers DC 24V 1=OK
      XT_DRP_OUT_PRT_3_CL : Bool;   // HDI def M 101.0: crystal drop out protection 3 closed (lower left side)
      XT_DRP_OUT_PRT_3_OP : Bool;   // HDI def M 101.1: crystal drop out protection 3 opened (lower left side)
      XT_DRP_OUT_PRT_4_CL : Bool;   // HDI def M 101.2: crystal drop out protection 4 closed (lower right side)
      XT_DRP_OUT_PRT_4_OP : Bool;   // HDI def M 101.3: crystal drop out protection 4 opened (lower right side)
      LS_XT_HDL_SW_UNLOCK : Bool;   // HDI def M 101.4: limit switch crystal handling swivel unlocked
      LS_XT_HDL_SW_LOCK : Bool;   // HDI def M 101.5: limit switch crystal handling swivel locked 145?
      LS_GCH_DOOR_OP : Bool;   // HDI def M 101.6: limit switch gate chamber door opened
      LS_GCH_DOOR_CL : Bool;   // HDI def M 101.7: limit switch gate chamber door closed
      MCC_CONTACT_XT : Bool;   // HDI def M 102.0: seed contact detection (xt isolated)
      OIL_LVL_XT_SFT : Bool;   // HDI def M 102.1: Crystal shaft min. oil level
      LS_XT_SFT_SRV_POS : Bool;   // HDI def M 102.2: limit switch crystal shaft service position
      LS_XT_TOP_POS : Bool;   // HDI def M 102.3: limit switch crystal shaft in top position
      SLS_TCH_LFT : Bool;   // HDI def M 102.4: Safety limit switch top chamber lift
      XT_ROT_CAM_TRG : Bool;   // HDI def M 102.5: limit switch xtal rotation camera trigger
      MP_ENB_K8 : Bool;   // HDI def M 102.6: Mobile panel agree button +K8
      MP_ENB_K9 : Bool;   // HDI def M 102.7: Mobile panel agree button +K9
      LS_V3_OP : Bool;   // HDI def M 103.0: valve position V3 open
      LS_V3_CL : Bool;   // HDI def M 103.1: Valve position V3 closed
      FDR_LS_V3_2_OP : Bool;   // HDI def M 103.2: valve position V3_2 open
      FDR_LS_V3_2_CL : Bool;   // HDI def M 103.3: Valve position V3_2 closed
      LSR_SEN_OBJ_DET : Bool;   // HDI def M 103.4: spare digital input
      SPARE_280_5 : Bool;   // HDI def M 103.5: spare digital input
      SPARE_280_6 : Bool;   // HDI def M 103.6: spare digital input
      SPARE_280_7 : Bool;   // HDI def M 103.7: spare digital input
      LS_V11_OP : Bool;   // HDI def M 89.3: V 11 open (isolation valve feeder)
      LS_V11_CL : Bool;   // HDI def M 89.4: V 11 closed (isolation valve feeder)
      FDR_HOP_CON : Bool;   // HDI def M 89.5: hopper connected to feeder
   END_VAR
BEGIN
END_DATA_BLOCK

DATA_BLOCK "IDO"   // DB897
{ S7_Optimized_Access := 'FALSE' }
VERSION : 0.0
// --------------------------------------------------------------------------------
// program:             IDO
// description :        automatically generated IDO
// name:                hp
// date        :        03.02.2021
// 
// revision:
// name:
// date:
//                     (c)CGS
// --------------------------------------------------------------------------------
   VAR
      HOR_OPP_K2 : Bool;   // HDO def M 136.0: Horn +K2
      LMP_RD_K2 : Bool;   // HDO def M 136.1: Lamp red +K2
      LMP_YE_K2 : Bool;   // HDO def M 136.2: Lamp yellow +K2
      LMP_GN_K2 : Bool;   // HDO def M 136.3: Lamp green +K2
      LMP_BU_K2 : Bool;   // HDO def M 136.4: Lamp blue +K2
      HOR_MAG_ACTIVE : Bool;   // HDO def M 136.5: Horn magnet active( Lift)
      LMP_MAG_ACTIVE : Bool;   // HDO def M 136.6: Lamp magnet active( Lift+ Field on)
      SPARE_16_7 : Bool;   // HDO def M 136.7: spare digital output
      P1_ON : Bool;   // HDO def M 137.0: Vacuum pump 1 on (furnace chamber)
      P3_ON : Bool;   // HDO def M 137.1: Vacuum pump 3 on (gate chamber)
      P2_ON : Bool;   // HDO def M 137.2: Vacuum pump 2 on (roots furnace chamber)
      P1_SEAL_GAS : Bool;   // HDO def M 137.3: Vacuum pump 1 seal gas on
      P3_SEAL_GAS : Bool;   // HDO def M 137.4: Vacuum pump 3 seal gas on
      HTR_PWR_ON : Bool;   // HDO def M 137.4: Heater power supply on
      V10 : Bool;   // HDO def M 137.6: Vacuum pump 1 secuvac valve V10 on
      MON_TMP_P2_RES : Bool;   // HDO def M 137.7: temperature monitoring pump 2 reset
      SPARE_18_0 : Bool;   // HDO def M 138.0: spare digital output
      SPARE_18_1 : Bool;   // HDO def M 138.1: spare digital output
      SPARE_18_2 : Bool;   // HDO def M 138.2: spare digital output
      SPARE_18_3 : Bool;   // HDO def M 138.3: spare digital output
      SPARE_18_4 : Bool;   // HDO def M 138.4: spare digital output
      SPARE_18_5 : Bool;   // HDO def M 138.5: spare digital output
      SPARE_18_6 : Bool;   // HDO def M 138.6: spare digital output
      SPARE_18_7 : Bool;   // HDO def M 138.7: spare digital output
      V1_OP : Bool;   // HDO def M 142.0: V1 open
      V1_CL : Bool;   // HDO def M 142.1: V1 close
      SPARE_32_2 : Bool;   // HDO def M 142.2: spare digital output
      SPARE_32_3 : Bool;   // HDO def M 142.3: spare digital output
      SPARE_32_4 : Bool;   // HDO def M 142.4: spare digital output
      CR_ROT_ENB : Bool;   // HDO def M 142.5: controller enable crucible rotation
      CR_LFT_ENB : Bool;   // HDO def M 142.6: controller enable crucible lift
      FU_FCB_HDL_ON : Bool;   // HDO def M 142.7: Frequency converter FCB handling on
      TEC_FLG_LFT_ENB : Bool;   // HDO def M 143.0: controller enable techn chamber lift
      FCH_LFT_ENB : Bool;   // HDO def M 143.1: controller enable lower chamber parts lift
      MAG_LFT_UP : Bool;   // HDO def M 143.2: Magnet lift drive upwards
      MAG_LFT_DN : Bool;   // HDO def M 143.3: Magnet lift drive downwards
      BRK_MAG_LFT : Bool;   // HDO def M 143.4: Brake magnet lift
      SPARE_33_5 : Bool;   // HDO def M 143.5: spare digital output
      SPARE_33_6 : Bool;   // HDO def M 143.6: spare digital output
      SPARE_33_7 : Bool;   // HDO def M 143.7: spare digital output
      V1_1_OP : Bool;   // HDO def M 144.0: V1.1 open
      V1_1_CL : Bool;   // HDO def M 144.1: V1.1 close
      SPARE_34_2 : Bool;   // HDO def M 144.2: spare digital output
      SPARE_34_3 : Bool;   // HDO def M 144.3: spare digital output
      SPARE_34_4 : Bool;   // HDO def M 144.4: spare digital output
      SPARE_34_5 : Bool;   // HDO def M 144.5: spare digital output
      SPARE_34_6 : Bool;   // HDO def M 144.6: spare digital output
      SPARE_34_7 : Bool;   // HDO def M 144.7: spare digital output
      ACC_SC_HTR_STR : Bool;   // HDO def M 146.0: ACC Heizung START
      ACC_SC_HTR_RST : Bool;   // HDO def M 146.1: ACC Heizung RESET
      ACC_SC_WTR_STR : Bool;   // HDO def M 146.2: ACC K黨lwasser START
      ACC_SC_WTR_RST : Bool;   // HDO def M 146.3: ACC K黨lwasser RESET
      ACC_ALM_LT_1 : Bool;   // HDO def M 146.4: ACC Blitzlicht Kasten
      ACC_ALM_SND_1 : Bool;   // HDO def M 146.5: ACC Sirene Kasten
      ACC_ALM_LT_2 : Bool;   // HDO def M 146.6: ACC Blitzlicht Bedienpult
      ACC_ALM_SND_2 : Bool;   // HDO def M 146.7: ACC Sirene Bedienpult
      FCH_HOOK_HOME : Bool;   // HDO def M 150.0: Valve block lower furnace chamber hook unlocking
      FCH_HOOK_WORK : Bool;   // HDO def M 150.1: Valve block lower furnace chamber hook locking
      UP_FCH_SW_BRK : Bool;   // HDO def M 150.2: Valve block upper chamber swivel release brake
      LO_FCH_SW_BRK : Bool;   // HDO def M 150.3: Valve block lower chamber swivel release brake
      TEC_FLG_SW_BRK : Bool;   // HDO def M 150.4: Valve block tech. flange swivel release brake
      V25 : Bool;   // HDO def M 150.5: Valve block argon inlet pressure storage tank, V25 open
      V2_1 : Bool;   // HDO def M 150.6: Valve block vacuum valve, V2.1 open
      V21 : Bool;   // HDO def M 150.7: Valve block air valve vacuum pipe, V21+V21.1 open
      V19 : Bool;   // HDO def M 151.0: Valve block extraktion valve filter, V19 open
      V20 : Bool;   // HDO def M 151.1: Valve block air valve filter, V20 open
      V22 : Bool;   // HDO def M 151.2: Valve block argon valve filter, V22 open
      V9_2 : Bool;   // HDO def M 151.3: Valve block ventiliation valve vaccum line gate, V9_2
      V22_1 : Bool;   // HDO def M 151.4: Valve block argon valve bypass filter, V22.1 open
      V3_4 : Bool;   // HDO def M 151.5: Valve block vacuum valve, V3.4 open
      V3_3 : Bool;   // HDO def M 151.6: Valve block vacuum valve, V3.3 open
      V2_11 : Bool;   // HDO def M 151.7: Valve block vacuum valve, V2.11 open
      P2_FU_ON : Bool;   // HDO def M 152.0: Frequency converter P2 start
      P2_FU_RES : Bool;   // HDO def M 152.1: Frequency converter P2 fault reset
      SPARE_144_2 : Bool;   // HDO def M 152.2: spare digital output
      SPARE_144_3 : Bool;   // HDO def M 152.3: spare digital output
      SPARE_144_4 : Bool;   // HDO def M 152.4: spare digital output
      SPARE_144_5 : Bool;   // HDO def M 152.5: spare digital output
      SPARE_144_6 : Bool;   // HDO def M 152.6: spare digital output
      SPARE_144_7 : Bool;   // HDO def M 152.7: spare digital output
      V4 : Bool;   // HDO def M 150.0: Valve block V4 valve argon gas inlet (gate chamber)
      V5 : Bool;   // HDO def M 150.1: Valve block V5 valve argon gas inlet controlled (gch)
      V6 : Bool;   // HDO def M 150.2: Valve block V6 valve argon gas inlet controlled (Fch)
      V3 : Bool;   // HDO def M 150.3: Valve block V3 vacuum valve (gate chamber)
      V3_2 : Bool;   // HDO def M 150.4: Valve block V3.2 vacuum valve feeder
      V24 : Bool;   // HDO def M 150.5: Valve block V24 valve argon gas inlet feeder
      XT_DRP_OUT_PRT_CL : Bool;   // HDO def M 150.6: Valve block close crystal drop out protection
      XT_DRP_OUT_PRT_OP : Bool;   // HDO def M 150.7: Valve block open crystal drop out protection
      TCH_SW_LOCK : Bool;   // HDO def M 151.0: Valve block top chamber swivel lock close
      TCH_SW_UNLOCK : Bool;   // HDO def M 151.1: Valve block top chamber swivel lock open
      GCH_SW_LOCK : Bool;   // HDO def M 151.2: Valve block gate chamber swivel lock close
      GCH_SW_UNLOCK : Bool;   // HDO def M 151.3: Valve block gate chamber swivel lock open
      XT_HDL_SW_LOCK : Bool;   // HDO def M 151.4: Valve block xtal handling swivel lock close (145?
      XT_HDL_SW_UNLOCK : Bool;   // HDO def M 151.5: Valve block xtal handling swivel lock open (145?
      FDR_V11_OP : Bool;   // HDO def M 151.6: Valve block open V11 (isolation valve feeder)
      FDR_V11_CL : Bool;   // HDO def M 151.7: Valve block close V11 (isolation valve feeder)
      FDR_V11_CVR_OP : Bool;   // HDO def M 152.0: Valve block open cover V11 (isolation valve feeder)
      FDR_V11_CVR_CL : Bool;   // HDO def M 152.1: Valve block close cover V11 (isolation valve feeder)
      SPARE_226_2 : Bool;   // HDO def M 152.2: Valve block spare output
      SPARE_226_3 : Bool;   // HDO def M 152.3: Valve block spare output
      SPARE_226_4 : Bool;   // HDO def M 152.4: Valve block spare output
      SPARE_226_5 : Bool;   // HDO def M 152.5: Valve block spare output
      SPARE_226_6 : Bool;   // HDO def M 152.6: Valve block spare output
      SPARE_226_7 : Bool;   // HDO def M 152.7: Valve block spare output
      HOR_OPP_K8 : Bool;   // HDO def M 160.0: Horn +K8
      LMP_RD_K8 : Bool;   // HDO def M 160.1: Lamp red +K8
      LMP_YE_K8 : Bool;   // HDO def M 160.2: Lamp yellow +K8
      LMP_GN_K8 : Bool;   // HDO def M 160.3: Lamp green +K8
      LMP_BU_K8 : Bool;   // HDO def M 160.4: Lamp blue +K8
      XT_ROT_ENB : Bool;   // HDO def M 160.5: controller enable crystal rotation
      XT_LFT_ENB : Bool;   // HDO def M 160.6: controller enable crystal lift
      XT_HDL_LFT_ENB : Bool;   // HDO def M 160.7: controller enable crystal handling lift
      XT_HDL_SW_ENB : Bool;   // HDO def M 161.0: controller enable crystal handling swivel
      FU_GCB_HDL_ON : Bool;   // HDO def M 161.1: Frequency converter GCB handling on
      LSR_SEN_PWR_ON : Bool;   // HDO def M 161.2: supply voltage for laser sensor on
      SPARE_273_3 : Bool;   // HDO def M 161.3: spare digital output
      SPARE_273_4 : Bool;   // HDO def M 161.4: spare digital output
      SPARE_273_5 : Bool;   // HDO def M 161.5: spare digital output
      XT_HDL_SLID_FW : Bool;   // HDO def M 161.6: Motor crystal handling slider forwards
      XT_HDL_SLID_BW : Bool;   // HDO def M 161.7: Motor crystal handling slider backwards
      XT_CLP_TILT_BW : Bool;   // HDO def M 163.0: Motor crystal clamp tilt backwards
      XT_CLP_TILT_FW : Bool;   // HDO def M 163.1: Motor crystal clamp tilt forwards (75?
      XT_CLP_TILT_BRK : Bool;   // HDO def M 163.2: Motor crystal clamp tilt brake
      XT_CLP_ABV_OP : Bool;   // HDO def M 163.3: Motor crystal clamp above open
      XT_CLP_ABV_CL : Bool;   // HDO def M 163.4: Motor crystal clamp above close
      XT_CLP_ABV_BRK : Bool;   // HDO def M 163.5: Brake crystal clamp above
      XT_CLP_ABV_RST : Bool;   // HDO def M 163.6: Reset controller crystal clamp above
      GCH_LFT_ENB : Bool;   // HDO def M 163.7: controller enable gate chamber lift
      XT_CLP_BLW_OP : Bool;   // HDO def M 164.0: Motor crystal clamp below open
      XT_CLP_BLW_CL : Bool;   // HDO def M 164.1: Motor crystal clamp below close
      XT_CLP_BLW_BRK : Bool;   // HDO def M 164.2: Brake crystal clamp below
      XT_CLP_BLW_RST : Bool;   // HDO def M 164.3: Reset controller crystal clamp below
      MCC_TEST_XT : Bool;   // HDO def M 164.4: seed contact detection test output ( xt isolated)
      MCC_ENB_XT : Bool;   // HDO def M 164.5: seed contact detection enable output (xt isolated)
      TCH_LFT_ENB : Bool;   // HDO def M 164.6: controller enable top chamber lift
      TCH_TILT_ENB : Bool;   // HDO def M 164.7: controller enable top chamber tilt
      GTE_V_LFT_ENB : Bool;   // HDO def M 165.0: controller enable gate valve lift
      GTE_V_SW_ENB : Bool;   // HDO def M 165.1: controller enable gate valve swivel
      BEL_LFT_ENB : Bool;   // HDO def M 165.2: controller enable gate bellow lift
      HOR_OPP_K9 : Bool;   // HDO def M 165.3: Horn +K9
      LMP_RD_K9 : Bool;   // HDO def M 165.4: Lamp red +K9
      LMP_YE_K9 : Bool;   // HDO def M 165.5: Lamp yellow +K9
      LMP_GN_K9 : Bool;   // HDO def M 165.6: Lamp green +K9
      LMP_BU_K9 : Bool;   // HDO def M 165.7: Lamp blue +K9
   END_VAR
BEGIN
END_DATA_BLOCK

DATA_BLOCK "CAI"   // DB898
{ S7_Optimized_Access := 'FALSE' }
VERSION : 0.0
// --------------------------------------------------------------------------------
// program:         CAI
// description :    configuration data for analog input [CAI.xxx]
//                  hardware_type   : int  - number of hardware i/o-type
//                  convert_type    : int  - number of linearization type
//                  description see in function PM_AI_CONVERT
//                  min_value       : real - min phys. value e.g. 0.0mm/min
//                  max_value       : real - max phys. value e.g. 8.0mm/min
//                  automatically generated CAI
// name:            hp
// date        :    03.02.2021
// 
// revision:
// name:
// date:
//                  (c)CGS
// --------------------------------------------------------------------------------
   VAR
      CONFIG_DATA : Array[1..60] of Struct
         hardware_type : Int;
         convert_type : Int;
         min_value : Real;
         max_value : Real;
      END_STRUCT;
   END_VAR
BEGIN
   CONFIG_DATA[1].hardware_type := 4;
   CONFIG_DATA[2].hardware_type := 4;
   CONFIG_DATA[3].hardware_type := 4;
   CONFIG_DATA[4].hardware_type := 4;
   CONFIG_DATA[5].hardware_type := 3;
   CONFIG_DATA[6].hardware_type := 3;
   CONFIG_DATA[7].hardware_type := 3;
   CONFIG_DATA[8].hardware_type := 4;
   CONFIG_DATA[9].hardware_type := 4;
   CONFIG_DATA[10].hardware_type := 4;
   CONFIG_DATA[11].hardware_type := 3;
   CONFIG_DATA[12].hardware_type := 3;
   CONFIG_DATA[13].hardware_type := 3;
   CONFIG_DATA[14].hardware_type := 3;
   CONFIG_DATA[15].hardware_type := 3;
   CONFIG_DATA[16].hardware_type := 3;
   CONFIG_DATA[1].convert_type := 2;
   CONFIG_DATA[2].convert_type := 2;
   CONFIG_DATA[3].convert_type := 2;
   CONFIG_DATA[4].convert_type := 2;
   CONFIG_DATA[5].convert_type := 2;
   CONFIG_DATA[6].convert_type := 2;
   CONFIG_DATA[7].convert_type := 2;
   CONFIG_DATA[8].convert_type := 9;
   CONFIG_DATA[9].convert_type := 9;
   CONFIG_DATA[10].convert_type := 2;
   CONFIG_DATA[11].convert_type := 2;
   CONFIG_DATA[12].convert_type := 2;
   CONFIG_DATA[13].convert_type := 2;
   CONFIG_DATA[14].convert_type := 2;
   CONFIG_DATA[15].convert_type := 2;
   CONFIG_DATA[16].convert_type := 2;
   CONFIG_DATA[5].min_value := 300.0;
   CONFIG_DATA[7].min_value := 900.0;
   CONFIG_DATA[1].max_value := 100.0;
   CONFIG_DATA[2].max_value := 100.0;
   CONFIG_DATA[3].max_value := 100.0;
   CONFIG_DATA[4].max_value := 100.0;
   CONFIG_DATA[5].max_value := 2000.0;
   CONFIG_DATA[6].max_value := 6.0;
   CONFIG_DATA[7].max_value := 1600.0;
   CONFIG_DATA[8].max_value := 1500.0;
   CONFIG_DATA[9].max_value := 1500.0;
   CONFIG_DATA[10].max_value := 100.0;
   CONFIG_DATA[11].max_value := 100.0;
   CONFIG_DATA[12].max_value := 10.0;
   CONFIG_DATA[13].max_value := 50.0;
   CONFIG_DATA[14].max_value := 50.0;
   CONFIG_DATA[15].max_value := 10.0;
   CONFIG_DATA[16].max_value := 700.0;
END_DATA_BLOCK

DATA_BLOCK "CAO"   // DB899
{ S7_Optimized_Access := 'FALSE' }
VERSION : 0.0
// --------------------------------------------------------------------------------
// program:         CAO
// description :    configuration data for analog input [CAI.xxx]
//                  hardware_type   : int  - number of hardware i/o-type
//                  convert_type    : int  - number of linearization type
//                  description see in function PM_AI_CONVERT
//                  min_value       : real - min phys. value e.g. 0.0mm/min
//                  max_value       : real - max phys. value e.g. 8.0mm/min
//                  automatically generated CAO
// name:            hp
// date        :    03.02.2021
// 
// revision:
// name:
// date:
//                  (c)CGS
// --------------------------------------------------------------------------------
   VAR
      CONFIG_DATA : Array[1..60] of Struct
         hardware_type : Int;
         convert_type : Int;
         min_value : Real;
         max_value : Real;
      END_STRUCT;
   END_VAR
BEGIN
   CONFIG_DATA[1].hardware_type := 3;
   CONFIG_DATA[2].hardware_type := 3;
   CONFIG_DATA[1].convert_type := 2;
   CONFIG_DATA[2].convert_type := 2;
   CONFIG_DATA[1].max_value := 100.0;
   CONFIG_DATA[2].max_value := 100.0;
END_DATA_BLOCK

DATA_BLOCK "CNF_XT_LFT_LZ950"   // DB904
{ S7_Optimized_Access := 'FALSE' }
VERSION : 0.0
// --------------------------------------------------------------------------------
//     program     :    CNF_XT_LFT_LZ950
//     description :    parameter for lenze-i950 if used for xtal-lift       
//     name        :    L. Vogel
//     date        :    06.06.2018
// 
//     revision    :    
//     name        :   
//     date        :    
//     
//                     (c)PVA CGS GMBH
//     --------------------------------------------------------------------------------
   VAR
      CTRL_ACTIV : Int := 1;   // 1 = controller installed
      PE_ADR : Int := 1632;   // start address for 3 words process data from controler
      PA_ADR : Int := 1632;   // start address for 3 words process data to controler
      GEAR_RATIO_Z : Real := 10.0;
      GEAR_RATIO_N : Real := 42.0;
      UNITS_PER_REV : Real := 10.0;
      FEED_CONST : Real := 0.2380952;   // 0.006613756; //1:42*10/1*1/36 10/42 = 0.2381
      MAX_SPEED : Real := 10.0;   // max. speed normal mode [mm/min] (C0011_N_MAX and gear ! )
      RATIO_FST_NRM : Real := 100.0;   // ratio fast/normal speed (C0941_CONV1_N / C0940_CONV1_D ! )
      RAMP_PITCH : Real := 1.0;
      Profil : Int := 1;   // Profil from 1-15 0 = No movement possible
      SEL_SPEED : Real := 8.0;   // selection speed
      SPARE : Real;
   END_VAR
BEGIN
END_DATA_BLOCK

DATA_BLOCK "CNF_XT_ROT_LZ950"   // DB905
{ S7_Optimized_Access := 'FALSE' }
VERSION : 0.0
// --------------------------------------------------------------------------------
//     program     :    CNF_XT_ROT_LZ950
//     description :    parameter for lenze-i950 if used for xtal-rotation       
//     name        :    L. Vogel
//     date        :    06.06.2018
// 
//     revision    :    
//     name        :   
//     date        :    
//     
//                     (c)PVA CGS GMBH
//     --------------------------------------------------------------------------------
   VAR
      CTRL_ACTIV : Int := 1;   // 1 = controller installed
      PE_ADR : Int := 1600;   // start address for 3 words process data from controler
      PA_ADR : Int := 1600;   // start address for 3 words process data to controler
      GEAR_RATIO_Z : Real := 1.0;
      GEAR_RATIO_N : Real := 100.0;
      UNITS_PER_REV : Real := 36.0;
      FEED_CONST : Real := 0.01;   // 0.00066127; //1:100*1/36 ;
      MAX_SPEED : Real := 20.0;   // max. speed normal mode [mm/min] (C0011_N_MAX and gear ! )
      RATIO_FST_NRM : Real := 1.0;   // ratio fast/normal speed (C0941_CONV1_N / C0940_CONV1_D ! )
      RAMP_PITCH : Real := 1.0;
      Profil : Int := 1;   // Profil from 1-15 0 = No movement possible
      SEL_SPEED : Real := 10.0;   // selection speed
      SPARE : Real;
   END_VAR
BEGIN
END_DATA_BLOCK

DATA_BLOCK "CNF_CR_LFT_LZ950"   // DB906
{ S7_Optimized_Access := 'FALSE' }
VERSION : 0.0
// --------------------------------------------------------------------------------
//     program     :    CNF_CR_LFT_LZ950
//     description :    parameter for lenze-i950 if used for crusible-lift       
//     name        :    L. Vogel
//     date        :    06.06.2018
// 
//     revision    :    
//     name        :   
//     date        :    
//     
//                     (c)PVA CGS GMBH
//     --------------------------------------------------------------------------------
   VAR
      CTRL_ACTIV : Int := 1;   // 1 = controller installed
      PE_ADR : Int := 672;   // start address for 3 words process data from controler
      PA_ADR : Int := 672;   // start address for 3 words process data to controler
      GEAR_RATIO_Z : Real := 4.0;
      GEAR_RATIO_N : Real := 42.0;
      UNITS_PER_REV : Real := 21.0;
      FEED_CONST : Real := 0.09494253;   // 1:42*4/1
      MAX_SPEED : Real := 2.6;   // max. speed normal mode [mm/min]
      RATIO_FST_NRM : Real := 100.0;   // ratio fast/normal speed
      RAMP_PITCH : Real := 1.0;
      Profil : Int := 1;   // Profil from 1-15 0 = No movement possible
      SEL_SPEED : Real := 2.0;   // selection speed
      SPARE : Real;
   END_VAR
BEGIN
END_DATA_BLOCK

DATA_BLOCK "CNF_CR_ROT_LZ950"   // DB907
{ S7_Optimized_Access := 'FALSE' }
VERSION : 0.0
// --------------------------------------------------------------------------------
//     program     :    CNF_CR_ROT_LZ950
//     description :    parameter for lenze-i950 if used for crusible-rotation       
//     name        :    L. Vogel
//     date        :    06.06.2018
// 
//     revision    :    
//     name        :   
//     date        :    
//     
//                     (c)PVA CGS GMBH
//     --------------------------------------------------------------------------------
   VAR
      CTRL_ACTIV : Int := 1;   // 1 = controller installed
      PE_ADR : Int := 640;   // start address for 3 words process data from controler
      PA_ADR : Int := 640;   // start address for 3 words process data to controler
      GEAR_RATIO_Z : Real := 1.0;
      GEAR_RATIO_N : Real := 100.0;
      UNITS_PER_REV : Real := 36.0;
      FEED_CONST : Real := 0.01;   // 0.00066127; //1:100*1/36 ;
      MAX_SPEED : Real := 20.0;   // max. speed normal mode [mm/min] (C0011_N_MAX and gear ! )
      RATIO_FST_NRM : Real := 1.0;   // ratio fast/normal speed (C0941_CONV1_N / C0940_CONV1_D ! )
      RAMP_PITCH : Real := 1.0;
      Profil : Int := 1;   // Profil from 1-15 0 = No movement possible
      SEL_SPEED : Real := 10.0;   // selection speed
      SPARE : Real;
   END_VAR
BEGIN
END_DATA_BLOCK

DATA_BLOCK "CNF_XT_HDL_LFT_LZ950"   // DB912
{ S7_Optimized_Access := 'FALSE' }
VERSION : 0.0
// --------------------------------------------------------------------------------
//     program     :    CNF_XT_HDL_LFT_LZ950
//     description :    parameter for lenze-i950 if used for crystal handling lift       
//     name        :    L. Vogel
//     date        :    06.06.2018
// 
//     revision    :    
//     name        :   
//     date        :    
//     
//                     (c)PVA CGS GMBH
//     --------------------------------------------------------------------------------
   VAR
      CTRL_ACTIV : Int := 1;   // 1 = controller installed
      PE_ADR : Int := 1664;   // start address for 3 words process data from controler
      PA_ADR : Int := 1664;   // start address for 3 words process data to controler
      GEAR_RATIO_Z : Real := 10.0;
      GEAR_RATIO_N : Real := 20.0;
      UNITS_PER_REV : Real := 42.0;
      FEED_CONST : Real := 0.5;   // 1:20*10/1*1/36;
      MAX_SPEED : Real := 1000.0;   // max. speed normal mode [mm/min] (C0011_N_MAX and gear ! )
      RATIO_FST_NRM : Real := 2.0;   // ratio fast/normal speed (C0941_CONV1_N / C0940_CONV1_D ! )
      RAMP_PITCH : Real := 1.0;
      Profil : Int := 1;   // Profil from 1-15 0 = No movement possible
      SEL_SPEED : Real := 500.0;   // selection speed
      SPARE : Real;
   END_VAR
BEGIN
END_DATA_BLOCK

DATA_BLOCK "CNF_XT_HDL_SW_LZ950"   // DB913
{ S7_Optimized_Access := 'FALSE' }
VERSION : 0.0
// --------------------------------------------------------------------------------
//     program     :    CNF_XT_HDL_SW_LZ950
//     description :    parameter for lenze-i950 if used for crystal handling swivel       
//     name        :    L. Vogel
//     date        :    06.06.2018
// 
//     revision    :    
//     name        :   
//     date        :    
//     
//                     (c)PVA CGS GMBH
//     --------------------------------------------------------------------------------
   VAR
      CTRL_ACTIV : Int := 1;   // 1 = controller installed
      PE_ADR : Int := 1696;   // start address for 3 words process data from controler
      PA_ADR : Int := 1696;   // start address for 3 words process data to controler
      GEAR_RATIO_Z : Real := 1.0;
      GEAR_RATIO_N : Real := 280.0;
      UNITS_PER_REV : Real := 36.0;
      FEED_CONST : Real := 1.285714;   // 1:280*360;
      MAX_SPEED : Real := 80.0;   // max. speed normal mode [mm/min] (C0011_N_MAX and gear ! )
      RATIO_FST_NRM : Real := 1.0;   // ratio fast/normal speed (C0941_CONV1_N / C0940_CONV1_D ! )
      RAMP_PITCH : Real := 1.0;
      Profil : Int := 1;   // Profil from 1-15 0 = No movement possible
      SEL_SPEED : Real := 80.0;   // selection speed
      SPARE : Real;
   END_VAR
BEGIN
END_DATA_BLOCK

DATA_BLOCK "CNF_BEL_LFT_LZ550"   // DB914
{ S7_Optimized_Access := 'FALSE' }
VERSION : 0.0
// --------------------------------------------------------------------------------
//     program     :    CNF_BEL_LFT_LZ550
//     description :    configuration data of lenze-i550 used for Gate chamber bellow lift       
//     name        :    John. Wang
//     date        :    26.10.2018
// 
//     revision    :    
//     name        :   
//     date        :    
//     
//                     (c)PVA CGS GmbH
//     --------------------------------------------------------------------------------
   VAR
      CTRL_ACTIV : Int := 1;   // 1 = controller installed
      PE_ADR : Int := 1888;   // input peripherie address
      PA_ADR : Int := 1888;   // output peripherie address
      SETP : Real := 30.0;   // set point lift speed in [Hz] (128#: 15.0 ; 100#: 30.0)
      SPARE : Real;
   END_VAR
BEGIN
END_DATA_BLOCK

DATA_BLOCK "CNF_GCH_LFT_LZ550"   // DB915
{ S7_Optimized_Access := 'FALSE' }
VERSION : 0.0
// --------------------------------------------------------------------------------
//     program     :    CNF_GCH_LFT_LZ550
//     description :    configuration data of lenze-i550 used for Gate chamber lift       
//     name        :    John. Wang
//     date        :    26.10.2018
// 
//     revision    :    
//     name        :   
//     date        :    
//     
//                     (c)PVA CGS GmbH
//     --------------------------------------------------------------------------------
   VAR
      CTRL_ACTIV : Int := 1;   // 1 = controller installed
      PE_ADR : Int := 1856;   // input peripherie address
      PA_ADR : Int := 1856;   // output peripherie address
      SETP : Real := 40.0;   // set point lift speed in [Hz]
      SPARE : Real;
   END_VAR
BEGIN
END_DATA_BLOCK

DATA_BLOCK "CNF_V7_LFT_LZ550"   // DB916
{ S7_Optimized_Access := 'FALSE' }
VERSION : 0.0
// --------------------------------------------------------------------------------
//     program     :    CNF_V7_LFT_LZ550
//     description :    configuration data of lenze-i550 for gate chamber valve lift                             
//     name        :    John. Wang
//     date        :    26.10.2018
// 
//     revision    :    
//     name        :   
//     date        :    
//     
//                     (c)PVA CGS GmbH
//     --------------------------------------------------------------------------------
   VAR
      CTRL_ACTIV : Int := 1;   // 1 = controller installed
      PE_ADR : Int := 1792;   // input peripherie address
      PA_ADR : Int := 1792;   // output peripherie address
      SETP : Real := 5.0;   // set point lift speed in [Hz]
      SPARE : Real;
   END_VAR
BEGIN
END_DATA_BLOCK

DATA_BLOCK "CNF_V7_SW_LZ550"   // DB917
{ S7_Optimized_Access := 'FALSE' }
VERSION : 0.0
// --------------------------------------------------------------------------------
//     program     :    CNF_V7_SW_LZ550
//     description :    configuration data of lenze-i550 for gate chamber valve swivel       
//     name        :    John. Wang
//     date        :    26.10.2018
// 
//     revision    :    
//     name        :   
//     date        :    
//     
//                     (c)PVA CGS GmbH
//     --------------------------------------------------------------------------------
   VAR
      CTRL_ACTIV : Int := 1;   // 1 = controller installed
      PE_ADR : Int := 1824;   // input peripherie address
      PA_ADR : Int := 1824;   // output peripherie address
      SETP : Real := 4.0;   // set point lift speed in [Hz] (128#:3.0 ; 100#:4.0)
      SPARE : Real;
   END_VAR
BEGIN
END_DATA_BLOCK

DATA_BLOCK "CNF_TCH_LFT_LZ550"   // DB918
{ S7_Optimized_Access := 'FALSE' }
VERSION : 0.0
// --------------------------------------------------------------------------------
//     program     :    CNF_TCH_LFT_LZ550
//     description :    configuration data of lenze-i550 for top chamber lift
//     name        :    John. Wang
//     date        :    26.10.2018
// 
//     revision    :    
//     name        :   
//     date        :    
//     
//                     (c)PVA CGS GmbH
//     --------------------------------------------------------------------------------
   VAR
      CTRL_ACTIV : Int := 1;   // 1 = controller installed
      PE_ADR : Int := 1760;   // input peripherie address
      PA_ADR : Int := 1760;   // output peripherie address
      SETP : Real := 30.0;   // set point lift speed in [Hz]
      SPARE : Real;
   END_VAR
BEGIN
END_DATA_BLOCK

DATA_BLOCK "CNF_TCH_TILT_LZ550"   // DB919
{ S7_Optimized_Access := 'FALSE' }
VERSION : 0.0
// --------------------------------------------------------------------------------
//     program     :    CNF_TCH_TILT_LZ550
//     description :    configuration data of lenze-i550 for top chamber tilt       
//     name        :    John. Wang
//     date        :    26.10.2018
// 
//     revision    :    
//     name        :   
//     date        :    
//     
//                     (c)PVA CGS GmbH
//     --------------------------------------------------------------------------------
   VAR
      CTRL_ACTIV : Int := 1;   // 1 = controller installed
      PE_ADR : Int := 1728;   // input peripherie address
      PA_ADR : Int := 1728;   // output peripherie address
      SETP : Real := 20.0;   // set point lift speed in [Hz] (128#: 10.0 ; 100#: 20.0)
      SPARE : Real;
   END_VAR
BEGIN
END_DATA_BLOCK

DATA_BLOCK "CNF_TEC_FLG_LFT_LZ550"   // DB920
{ S7_Optimized_Access := 'FALSE' }
VERSION : 0.0
// --------------------------------------------------------------------------------
//     program     :    CNF_TEC_FLG_LFT_LZ550
//     description :    configuration data of lenze-i550 for technologie flange lift       
//     name        :    John. Wang
//     date        :    26.10.2018
// 
//     revision    :    
//     name        :   
//     date        : 
//     
//                     (c)PVA CGS GmbH
//     --------------------------------------------------------------------------------
   VAR
      CTRL_ACTIV : Int := 1;   // 1 = controller installed
      PE_ADR : Int := 704;   // input peripherie address
      PA_ADR : Int := 704;   // output peripherie address
      SETP : Real := 15.0;   // set point lift speed in [Hz]
      SETP_FST : Real := 25.0;
   END_VAR
BEGIN
END_DATA_BLOCK

DATA_BLOCK "CNF_FCH_LFT_LZ550"   // DB921
{ S7_Optimized_Access := 'FALSE' }
VERSION : 0.0
// --------------------------------------------------------------------------------
//     program     :    CNF_FCH_LFT_LZ550
//     description :    configuration data of lenze-i550 for upper furnace chamber lift       
//     name        :    John. Wang
//     date        :    26.10.2018
// 
//     revision    :    
//     name        :   
//     date        :    
//     
//                     (c)PVA CGS GmbH
//     --------------------------------------------------------------------------------
   VAR
      CTRL_ACTIV : Int := 1;   // 1 = controller installed
      PE_ADR : Int := 736;   // input peripherie address
      PA_ADR : Int := 736;   // output peripherie address
      SETP : Real := 20.0;   // set point lift speed in [Hz]
      SETP_FST : Real := 30.0;
   END_VAR
BEGIN
END_DATA_BLOCK

DATA_BLOCK "GLOBAL_DIAG_PN"   // DB1000
{ S7_Optimized_Access := 'FALSE' }
VERSION : 0.0
// --------------------------------------------------------------------------------
//     program     :    GLOBAL_DIAG_PN
//     description :    data block for l2 net diagnosis        
//     name:            L. Vogel
//     date        :    12.10.2018
// 
//     revision    :   
//     name        :
//     date        :    
//                     (c)PVA CGS GmbH
//     --------------------------------------------------------------------------------
   VAR
      index : Word;
      Device_status : Array[0..2047] of Bool;
      Device_spare : Array[1..10] of Byte;
      RET_VAL_DP : Int;
      BUSY_DP : Bool;
      RET_VAL_PNIO : Int;
      BUSY_PNIO : Bool;
      SPARE_DATA : Array[1..10] of Byte;
      SSL_HEADER : Struct
         LENTHDR : Word;
         N_DR : Word;
      END_STRUCT;
      SPARE_290 : Array[1..10] of Byte;
   END_VAR
BEGIN
END_DATA_BLOCK

DATA_BLOCK "PAR_CTRL_GAP_GN"   // DB1100
{ S7_Optimized_Access := 'FALSE' }
VERSION : 0.0
BEGIN
END_DATA_BLOCK

DATA_BLOCK "PAR_CTRL_GAP_TI"   // DB1101
{ S7_Optimized_Access := 'FALSE' }
VERSION : 0.0
BEGIN
END_DATA_BLOCK

DATA_BLOCK "PAR_CTRL_GAP_TD"   // DB1102
{ S7_Optimized_Access := 'FALSE' }
VERSION : 0.0
BEGIN
END_DATA_BLOCK

DATA_BLOCK "PAR_CTRL_GAP_T1"   // DB1103
{ S7_Optimized_Access := 'FALSE' }
VERSION : 0.0
BEGIN
END_DATA_BLOCK

DATA_BLOCK "PAR_CTL_OFFS_SPD_GN"   // DB1104
{ S7_Optimized_Access := 'FALSE' }
VERSION : 0.0
BEGIN
END_DATA_BLOCK

DATA_BLOCK "PAR_CTL_OFFS_SPD_TI"   // DB1105
{ S7_Optimized_Access := 'FALSE' }
VERSION : 0.0
BEGIN
END_DATA_BLOCK

DATA_BLOCK "PAR_CTL_OFFS_SPD_TD"   // DB1106
{ S7_Optimized_Access := 'FALSE' }
VERSION : 0.0
BEGIN
END_DATA_BLOCK

DATA_BLOCK "PAR_CTL_OFFS_SPD_T1"   // DB1107
{ S7_Optimized_Access := 'FALSE' }
VERSION : 0.0
BEGIN
END_DATA_BLOCK

DATA_BLOCK "PAR_CTL_OFFS_AVR_GN"   // DB1108
{ S7_Optimized_Access := 'FALSE' }
VERSION : 0.0
BEGIN
END_DATA_BLOCK

DATA_BLOCK "PAR_CTL_OFFS_AVR_TI"   // DB1109
{ S7_Optimized_Access := 'FALSE' }
VERSION : 0.0
BEGIN
END_DATA_BLOCK

DATA_BLOCK "PAR_CTL_OFFS_AVR_TD"   // DB1110
{ S7_Optimized_Access := 'FALSE' }
VERSION : 0.0
BEGIN
END_DATA_BLOCK

DATA_BLOCK "PAR_CTL_OFFS_AVR_T1"   // DB1111
{ S7_Optimized_Access := 'FALSE' }
VERSION : 0.0
BEGIN
END_DATA_BLOCK

DATA_BLOCK "PAR_SCAM_CTR_X_POS"   // DB1112
{ S7_Optimized_Access := 'FALSE' }
VERSION : 0.0
BEGIN
END_DATA_BLOCK

DATA_BLOCK "PAR_SCAM_CTR_Y_POS"   // DB1113
{ S7_Optimized_Access := 'FALSE' }
VERSION : 0.0
BEGIN
END_DATA_BLOCK

DATA_BLOCK "PAR_CAM_2_THR"   // DB1114
{ S7_Optimized_Access := 'FALSE' }
VERSION : 0.0
BEGIN
END_DATA_BLOCK

DATA_BLOCK "SEND_MES"   // DB1200
{ S7_Optimized_Access := 'FALSE' }
VERSION : 0.0
// --------------------------------------------------------------------------------
//     program     :    SEND_MES
//     description :    data for communication to MES  
//     name        :    L. Vogel
//     date        :    12.02.2019
// 
//     revision    :
//     name        :
//     date        :    
//                     (c)PVA CGS GMBH
//     --------------------------------------------------------------------------------
   VAR
      Header : Array[1..32] of Bool;
      MachineNo : Int;
      MachineStatus : Int;
      ACT_PROCESS : Int;   // actual process phase
      Timestamp : Date_And_Time;
      User_Name : String[30];   // actual recipe name
      ACT_RCP_NAME : String[200];   // actual recipe name
      ACT_INGOT_ID : String[200];   // actual ingot number (ID)
      ACT_CHARGE_ID : String[30];   // actual charge number (ID)
      ACT_CRU_ID : String[30];   // actual cruible number (ID)
      SPARE : Array[1..30] of Byte;
      ACT_XT_SPD : Real;   // actual crystal pull speed
      ACT_XT_ROT : Real;   // actual crystal rotation speed
      ACT_XT_POS : Real;   // actual crystal lift position
      ACT_CR_SPD : Real;   // actual crucible lift speed
      ACT_CR_ROT : Real;   // actual crucible rotation speed
      ACT_CR_POS : Real;   // actual crucible lift position
      ACT_HTR_1_PWR : Real;   // actual power main heater
      ACT_HTR_1_TMP : Real;   // actual temperature main heater
      ACT_HTR_2_PWR : Real;   // actual power bottom heater
      ACT_MAG_1_CUR : Real;   // actual current magnet 1
      ACT_MAG_2_CUR : Real;   // actual current magnet 2
      ACT_GAS_1_FLW : Real;   // actual gas flow 1
      ACT_GAS_2_FLW : Real;   // actual gas flow 1
      ACT_TOT_XT_LGH : Real;   // actual total crystal lenght (neck, shoulder, body, endcone)
      ACT_PRS_CLF : Real;   // actual pressure furnace
      ACT_PRS_CGT : Real;   // actual pressure gate
      ACT_XT_DIA : Real;   // actual crystal diameter
      ACT_XT_LEN_MM : Real;   // actual crystal length/phase
      Spare_432 : Real;
      Spare_436 : Real;
      CHARGE_WGT : Real;   // actual charge weight (Recipe)
      CRU_QRZ_WALL_THICKN : Real;   // actual crucible quartz wall thickness (Recipe)
      CRU_QRZ_BOT_THICKN : Real;   // actual crucible quartz bottom thickness (Recipe)
      CRU_QRZ_TRANS_RAD : Real;   // actual crucible quartz transition radius (Recipe)
      CRU_GRAPH_BOT_RAD : Real;   // actual crucible graphite bottom radius (Recipe)
      CRU_GRAPH_INNER_DIA : Real;   // actual crucible graphite inner diameter (Recipe)
      Spare_464 : Real;
      Spare_468 : Real;
      Spare_472 : Real;
      Spare_476 : Real;
      FAULT : Array[0..10] of Int;
   END_VAR
BEGIN
END_DATA_BLOCK

DATA_BLOCK "RECV_MES"   // DB1201
{ S7_Optimized_Access := 'FALSE' }
VERSION : 0.0
// --------------------------------------------------------------------------------
//     program     :    RECV_MES
//     description :    data for communication from MES  
//     name        :    L. Vogel
//     date        :    12.02.2019
// 
//     revision    :
//     name        :
//     date        :    
//                     (c)PVA CGS GMBH
//     --------------------------------------------------------------------------------
   VAR
      Header : DWord;
      ACT_RCP_NAME : String[200];   // actual recipe name
      ACT_INGOT_ID : String[200];   // actual ingot number (ID)
      ACT_CHARGE_ID : String[30];   // actual charge number (ID)
      ACT_CRU_ID : String[30];   // actual cruible number (ID)
      SPARE : Array[1..30] of Byte;
   END_VAR
BEGIN
END_DATA_BLOCK

FUNCTION_BLOCK "PM_DI"   // FB17, SCL
{ S7_Optimized_Access := 'FALSE' }
VERSION : 0.0
// --------------------------------------------------------------------------------
//     program:         PM_DI
//     description :    automatically generated PM_DI
//     name:            hp
//     date        :    03.02.2021
// 
//     revision:
//     name:
//     Date:
//                     (c)CGS
//     --------------------------------------------------------------------------------
   VAR
      y : Bool;
      count : Int := 8;
   END_VAR
   VAR_TEMP
      x : Bool;
   END_VAR
BEGIN


   IF "SY".SIM_ON AND NOT "SY".SRM_ON THEN

       "PDI".CB_FLT_DC24V_K2 := "SDI".CB_FLT_DC24V_K2 XOR "IDI".CB_FLT_DC24V_K2;
       "PDI".CB_FLT_AC400V_K2 := "SDI".CB_FLT_AC400V_K2 XOR "IDI".CB_FLT_AC400V_K2;
       "PDI".SPARE_16_2 := "SDI".SPARE_16_2 XOR "IDI".SPARE_16_2;
       "PDI".CB_FLT_AC230V := "SDI".CB_FLT_AC230V XOR "IDI".CB_FLT_AC230V;
       "PDI".SPARE_16_4 := "SDI".SPARE_16_4 XOR "IDI".SPARE_16_4;
       "PDI".SPARE_16_5 := "SDI".SPARE_16_5 XOR "IDI".SPARE_16_5;
       "PDI".SPARE_16_6 := "SDI".SPARE_16_6 XOR "IDI".SPARE_16_6;
       "PDI".SPARE_16_7 := "SDI".SPARE_16_7 XOR "IDI".SPARE_16_7;
       "PDI".SPARE_17_0 := "SDI".SPARE_17_0 XOR "IDI".SPARE_17_0;
       "PDI".UPS_24V_ALM := "SDI".UPS_24V_ALM XOR "IDI".UPS_24V_ALM;
       "PDI".UPS_24V_NRM := "SDI".UPS_24V_NRM XOR "IDI".UPS_24V_NRM;
       "PDI".EMO := "SDI".EMO XOR "IDI".EMO;
       "PDI".EMS := "SDI".EMS XOR "IDI".EMS;
       "PDI".SPARE_17_5 := "SDI".SPARE_17_5 XOR "IDI".SPARE_17_5;
       "PDI".SPARE_17_6 := "SDI".SPARE_17_6 XOR "IDI".SPARE_17_6;
       "PDI".SPARE_17_7 := "SDI".SPARE_17_7 XOR "IDI".SPARE_17_7;
       "PDI".P1_WRN := "SDI".P1_WRN XOR "IDI".P1_WRN;
       "PDI".P1_FLT := "SDI".P1_FLT XOR "IDI".P1_FLT;
       "PDI".P1_IS_ON := "SDI".P1_IS_ON XOR "IDI".P1_IS_ON;
       "PDI".P1_WD := "SDI".P1_WD XOR "IDI".P1_WD;
       "PDI".FIL_APS := "SDI".FIL_APS XOR "IDI".FIL_APS;
       "PDI".MON_TMP_P2 := "SDI".MON_TMP_P2 XOR "IDI".MON_TMP_P2;
       "PDI".MON_TMP_P1 := "SDI".MON_TMP_P1 XOR "IDI".MON_TMP_P1;
       "PDI".SPARE_18_7 := "SDI".SPARE_18_7 XOR "IDI".SPARE_18_7;
       "PDI".FCH_LFT_SDL_NUT := "SDI".FCH_LFT_SDL_NUT XOR "IDI".FCH_LFT_SDL_NUT;
       "PDI".LS_FCH_LFT_DN := "SDI".LS_FCH_LFT_DN XOR "IDI".LS_FCH_LFT_DN;
       "PDI".LS_FCH_HOOK_WORK := "SDI".LS_FCH_HOOK_WORK XOR "IDI".LS_FCH_HOOK_WORK;
       "PDI".LS_FCH_HOOK_HOME := "SDI".LS_FCH_HOOK_HOME XOR "IDI".LS_FCH_HOOK_HOME;
       "PDI".LS_TEC_FLG_DN := "SDI".LS_TEC_FLG_DN XOR "IDI".LS_TEC_FLG_DN;
       "PDI".TEC_FLG_SDL_NUT := "SDI".TEC_FLG_SDL_NUT XOR "IDI".TEC_FLG_SDL_NUT;
       "PDI".LS_V11_COV_OP := "SDI".LS_V11_COV_OP XOR "IDI".LS_V11_COV_OP;
       "PDI".LS_V11_COV_CL := "SDI".LS_V11_COV_CL XOR "IDI".LS_V11_COV_CL;
       "PDI".GCH_APS := "SDI".GCH_APS XOR "IDI".GCH_APS;
       "PDI".FCH_APS := "SDI".FCH_APS XOR "IDI".FCH_APS;
       "PDI".FDR_APS := "SDI".FDR_APS XOR "IDI".FDR_APS;
       "PDI".FIL_2_APS := "SDI".FIL_2_APS XOR "IDI".FIL_2_APS;
       "PDI".SPARE_33_4 := "SDI".SPARE_33_4 XOR "IDI".SPARE_33_4;
       "PDI".SPARE_33_5 := "SDI".SPARE_33_5 XOR "IDI".SPARE_33_5;
       "PDI".LS_V2_1_OP := "SDI".LS_V2_1_OP XOR "IDI".LS_V2_1_OP;
       "PDI".LS_V2_1_CL := "SDI".LS_V2_1_CL XOR "IDI".LS_V2_1_CL;
       "PDI".CB_FLT_AC400V_K5 := "SDI".CB_FLT_AC400V_K5 XOR "IDI".CB_FLT_AC400V_K5;
       "PDI".CB_FLT_DC24V_K5 := "SDI".CB_FLT_DC24V_K5 XOR "IDI".CB_FLT_DC24V_K5;
       "PDI".LS_MAG_LFT_UP := "SDI".LS_MAG_LFT_UP XOR "IDI".LS_MAG_LFT_UP;
       "PDI".LS_MAG_LFT_DN := "SDI".LS_MAG_LFT_DN XOR "IDI".LS_MAG_LFT_DN;
       "PDI".SLS_MAG_LFT := "SDI".SLS_MAG_LFT XOR "IDI".SLS_MAG_LFT;
       "PDI".MAG_LFT_SDL_NUT1 := "SDI".MAG_LFT_SDL_NUT1 XOR "IDI".MAG_LFT_SDL_NUT1;
       "PDI".MAG_LFT_SDL_NUT2 := "SDI".MAG_LFT_SDL_NUT2 XOR "IDI".MAG_LFT_SDL_NUT2;
       "PDI".MAG_LFT_SDL_NUT3 := "SDI".MAG_LFT_SDL_NUT3 XOR "IDI".MAG_LFT_SDL_NUT3;
       "PDI".OIL_LVL_CR_SFT := "SDI".OIL_LVL_CR_SFT XOR "IDI".OIL_LVL_CR_SFT;
       "PDI".LS_V1_OP := "SDI".LS_V1_OP XOR "IDI".LS_V1_OP;
       "PDI".LS_V1_CL := "SDI".LS_V1_CL XOR "IDI".LS_V1_CL;
       "PDI".MP_ENB_K5 := "SDI".MP_ENB_K5 XOR "IDI".MP_ENB_K5;
       "PDI".SLS_TEC_FLG_LFT := "SDI".SLS_TEC_FLG_LFT XOR "IDI".SLS_TEC_FLG_LFT;
       "PDI".SLS_FCH_LFT := "SDI".SLS_FCH_LFT XOR "IDI".SLS_FCH_LFT;
       "PDI".COMP_AIR_OK := "SDI".COMP_AIR_OK XOR "IDI".COMP_AIR_OK;
       "PDI".COMP_AIR_2_OK := "SDI".COMP_AIR_2_OK XOR "IDI".COMP_AIR_2_OK;
       "PDI".LS_V1_1_CL := "SDI".LS_V1_1_CL XOR "IDI".LS_V1_1_CL;
       "PDI".LS_V1_1_OP := "SDI".LS_V1_1_OP XOR "IDI".LS_V1_1_OP;
       "PDI".LS_V3_4_OP := "SDI".LS_V3_4_OP XOR "IDI".LS_V3_4_OP;
       "PDI".LS_V3_4_CL := "SDI".LS_V3_4_CL XOR "IDI".LS_V3_4_CL;
       "PDI".LS_V3_3_OP := "SDI".LS_V3_3_OP XOR "IDI".LS_V3_3_OP;
       "PDI".LS_V3_3_CL := "SDI".LS_V3_3_CL XOR "IDI".LS_V3_3_CL;
       "PDI".LS_V2_11_OP := "SDI".LS_V2_11_OP XOR "IDI".LS_V2_11_OP;
       "PDI".LS_V2_11_CL := "SDI".LS_V2_11_CL XOR "IDI".LS_V2_11_CL;
       "PDI".ACC_FCH_OV_PRS_1 := "SDI".ACC_FCH_OV_PRS_1 XOR "IDI".ACC_FCH_OV_PRS_1;
       "PDI".ACC_FCH_OV_PRS_2 := "SDI".ACC_FCH_OV_PRS_2 XOR "IDI".ACC_FCH_OV_PRS_2;
       "PDI".SPARE_48_2 := "SDI".SPARE_48_2 XOR "IDI".SPARE_48_2;
       "PDI".ACC_WTR_FLW_OUT_OK := "SDI".ACC_WTR_FLW_OUT_OK XOR "IDI".ACC_WTR_FLW_OUT_OK;
       "PDI".ACC_WTR_FLW_IN_OK := "SDI".ACC_WTR_FLW_IN_OK XOR "IDI".ACC_WTR_FLW_IN_OK;
       "PDI".ACC_WTR_TMP_OUT_OK := "SDI".ACC_WTR_TMP_OUT_OK XOR "IDI".ACC_WTR_TMP_OUT_OK;
       "PDI".OV_PRS_1_FLT := "SDI".OV_PRS_1_FLT XOR "IDI".OV_PRS_1_FLT;
       "PDI".OV_PRS_2_FLT := "SDI".OV_PRS_2_FLT XOR "IDI".OV_PRS_2_FLT;
       "PDI".ACC_SC_WTR_OK := "SDI".ACC_SC_WTR_OK XOR "IDI".ACC_SC_WTR_OK;
       "PDI".ACC_SC_WTR_ATV := "SDI".ACC_SC_WTR_ATV XOR "IDI".ACC_SC_WTR_ATV;
       "PDI".ACC_SC_HTR_OK := "SDI".ACC_SC_HTR_OK XOR "IDI".ACC_SC_HTR_OK;
       "PDI".ACC_SC_HTR_ATV := "SDI".ACC_SC_HTR_ATV XOR "IDI".ACC_SC_HTR_ATV;
       "PDI".ACC_KEY_RST := "SDI".ACC_KEY_RST XOR "IDI".ACC_KEY_RST;
       "PDI".ACC_CB_FLT_DC24V := "SDI".ACC_CB_FLT_DC24V XOR "IDI".ACC_CB_FLT_DC24V;
       "PDI".ACC_UPS_24V_ALM := "SDI".ACC_UPS_24V_ALM XOR "IDI".ACC_UPS_24V_ALM;
       "PDI".ACC_UPS_24V_NRM := "SDI".ACC_UPS_24V_NRM XOR "IDI".ACC_UPS_24V_NRM;
       "PDI".DPH_RPT_DET_OK := "SDI".DPH_RPT_DET_OK XOR "IDI".DPH_RPT_DET_OK;
       "PDI".ACC_CB_FLT_AC230V := "SDI".ACC_CB_FLT_AC230V XOR "IDI".ACC_CB_FLT_AC230V;
       "PDI".SPARE_90_2 := "SDI".SPARE_90_2 XOR "IDI".SPARE_90_2;
       "PDI".SPARE_90_3 := "SDI".SPARE_90_3 XOR "IDI".SPARE_90_3;
       "PDI".SPARE_90_4 := "SDI".SPARE_90_4 XOR "IDI".SPARE_90_4;
       "PDI".SPARE_90_5 := "SDI".SPARE_90_5 XOR "IDI".SPARE_90_5;
       "PDI".SPARE_90_6 := "SDI".SPARE_90_6 XOR "IDI".SPARE_90_6;
       "PDI".SPARE_90_7 := "SDI".SPARE_90_7 XOR "IDI".SPARE_90_7;
       "PDI".FU_P2_RDY := "SDI".FU_P2_RDY XOR "IDI".FU_P2_RDY;
       "PDI".SPARE_144_1 := "SDI".SPARE_144_1 XOR "IDI".SPARE_144_1;
       "PDI".LS_GCH_UP := "SDI".LS_GCH_UP XOR "IDI".LS_GCH_UP;
       "PDI".LS_GCH_DN := "SDI".LS_GCH_DN XOR "IDI".LS_GCH_DN;
       "PDI".LS_GCH_SW_IN := "SDI".LS_GCH_SW_IN XOR "IDI".LS_GCH_SW_IN;
       "PDI".LS_GCH_SW_CLN := "SDI".LS_GCH_SW_CLN XOR "IDI".LS_GCH_SW_CLN;
       "PDI".LS_GCH_SW_OUT := "SDI".LS_GCH_SW_OUT XOR "IDI".LS_GCH_SW_OUT;
       "PDI".LS_GCH_SW_LOCK := "SDI".LS_GCH_SW_LOCK XOR "IDI".LS_GCH_SW_LOCK;
       "PDI".SLS_GCH_LFT := "SDI".SLS_GCH_LFT XOR "IDI".SLS_GCH_LFT;
       "PDI".LS_TCH_UP := "SDI".LS_TCH_UP XOR "IDI".LS_TCH_UP;
       "PDI".LS_TCH_DN := "SDI".LS_TCH_DN XOR "IDI".LS_TCH_DN;
       "PDI".LS_TCH_SW_IN := "SDI".LS_TCH_SW_IN XOR "IDI".LS_TCH_SW_IN;
       "PDI".LS_TCH_SW_CLN := "SDI".LS_TCH_SW_CLN XOR "IDI".LS_TCH_SW_CLN;
       "PDI".LS_TCH_SW_OUT := "SDI".LS_TCH_SW_OUT XOR "IDI".LS_TCH_SW_OUT;
       "PDI".LS_TCH_SW_LOCK := "SDI".LS_TCH_SW_LOCK XOR "IDI".LS_TCH_SW_LOCK;
       "PDI".LS_TCH_TILT_0 := "SDI".LS_TCH_TILT_0 XOR "IDI".LS_TCH_TILT_0;
       "PDI".LS_TCH_TILT_30 := "SDI".LS_TCH_TILT_30 XOR "IDI".LS_TCH_TILT_30;
       "PDI".KEY_XT_LFT_SRV := "SDI".KEY_XT_LFT_SRV XOR "IDI".KEY_XT_LFT_SRV;
       "PDI".LS_V7_UP := "SDI".LS_V7_UP XOR "IDI".LS_V7_UP;
       "PDI".LS_V7_DN := "SDI".LS_V7_DN XOR "IDI".LS_V7_DN;
       "PDI".LS_V7_SW_IN := "SDI".LS_V7_SW_IN XOR "IDI".LS_V7_SW_IN;
       "PDI".LS_V7_SW_OUT := "SDI".LS_V7_SW_OUT XOR "IDI".LS_V7_SW_OUT;
       "PDI".LS_V7_FLP_OP := "SDI".LS_V7_FLP_OP XOR "IDI".LS_V7_FLP_OP;
       "PDI".LS_V7_CLN_POS := "SDI".LS_V7_CLN_POS XOR "IDI".LS_V7_CLN_POS;
       "PDI".LS_GCH_BEL_UP := "SDI".LS_GCH_BEL_UP XOR "IDI".LS_GCH_BEL_UP;
       "PDI".LS_GCH_BEL_DN := "SDI".LS_GCH_BEL_DN XOR "IDI".LS_GCH_BEL_DN;
       "PDI".LS_XT_SLID_BW := "SDI".LS_XT_SLID_BW XOR "IDI".LS_XT_SLID_BW;
       "PDI".LS_XT_SLID_FW := "SDI".LS_XT_SLID_FW XOR "IDI".LS_XT_SLID_FW;
       "PDI".LS_XT_SLID_MID := "SDI".LS_XT_SLID_MID XOR "IDI".LS_XT_SLID_MID;
       "PDI".LS_XT_CLP_CON := "SDI".LS_XT_CLP_CON XOR "IDI".LS_XT_CLP_CON;
       "PDI".LS_XT_TILT_90 := "SDI".LS_XT_TILT_90 XOR "IDI".LS_XT_TILT_90;
       "PDI".LS_XT_TILT_75 := "SDI".LS_XT_TILT_75 XOR "IDI".LS_XT_TILT_75;
       "PDI".LS_UP_XT_CLP_FLT := "SDI".LS_UP_XT_CLP_FLT XOR "IDI".LS_UP_XT_CLP_FLT;
       "PDI".SPARE_275_7 := "SDI".SPARE_275_7 XOR "IDI".SPARE_275_7;
       "PDI".LS_UP_XT_CLP_OP := "SDI".LS_UP_XT_CLP_OP XOR "IDI".LS_UP_XT_CLP_OP;
       "PDI".LS_UP_XT_CLP_CL := "SDI".LS_UP_XT_CLP_CL XOR "IDI".LS_UP_XT_CLP_CL;
       "PDI".LS_UP_XT_CLP_SAVE := "SDI".LS_UP_XT_CLP_SAVE XOR "IDI".LS_UP_XT_CLP_SAVE;
       "PDI".LS_UP_XT_CLP_PLATE := "SDI".LS_UP_XT_CLP_PLATE XOR "IDI".LS_UP_XT_CLP_PLATE;
       "PDI".LS_LO_XT_CLP_FLT := "SDI".LS_LO_XT_CLP_FLT XOR "IDI".LS_LO_XT_CLP_FLT;
       "PDI".LS_LO_XT_CLP_OP := "SDI".LS_LO_XT_CLP_OP XOR "IDI".LS_LO_XT_CLP_OP;
       "PDI".LS_LO_XT_CLP_CL := "SDI".LS_LO_XT_CLP_CL XOR "IDI".LS_LO_XT_CLP_CL;
       "PDI".LS_LO_XT_CLP_SAVE := "SDI".LS_LO_XT_CLP_SAVE XOR "IDI".LS_LO_XT_CLP_SAVE;
       "PDI".LS_LO_XT_CLP_PLATE := "SDI".LS_LO_XT_CLP_PLATE XOR "IDI".LS_LO_XT_CLP_PLATE;
       "PDI".LS_HOI_TOOL_INST := "SDI".LS_HOI_TOOL_INST XOR "IDI".LS_HOI_TOOL_INST;
       "PDI".XT_DRP_OUT_PRT_1_CL := "SDI".XT_DRP_OUT_PRT_1_CL XOR "IDI".XT_DRP_OUT_PRT_1_CL;
       "PDI".XT_DRP_OUT_PRT_1_OP := "SDI".XT_DRP_OUT_PRT_1_OP XOR "IDI".XT_DRP_OUT_PRT_1_OP;
       "PDI".XT_DRP_OUT_PRT_2_CL := "SDI".XT_DRP_OUT_PRT_2_CL XOR "IDI".XT_DRP_OUT_PRT_2_CL;
       "PDI".XT_DRP_OUT_PRT_2_OP := "SDI".XT_DRP_OUT_PRT_2_OP XOR "IDI".XT_DRP_OUT_PRT_2_OP;
       "PDI".CB_FLT_AC400V_K8 := "SDI".CB_FLT_AC400V_K8 XOR "IDI".CB_FLT_AC400V_K8;
       "PDI".CB_FLT_DC24V_K8 := "SDI".CB_FLT_DC24V_K8 XOR "IDI".CB_FLT_DC24V_K8;
       "PDI".XT_DRP_OUT_PRT_3_CL := "SDI".XT_DRP_OUT_PRT_3_CL XOR "IDI".XT_DRP_OUT_PRT_3_CL;
       "PDI".XT_DRP_OUT_PRT_3_OP := "SDI".XT_DRP_OUT_PRT_3_OP XOR "IDI".XT_DRP_OUT_PRT_3_OP;
       "PDI".XT_DRP_OUT_PRT_4_CL := "SDI".XT_DRP_OUT_PRT_4_CL XOR "IDI".XT_DRP_OUT_PRT_4_CL;
       "PDI".XT_DRP_OUT_PRT_4_OP := "SDI".XT_DRP_OUT_PRT_4_OP XOR "IDI".XT_DRP_OUT_PRT_4_OP;
       "PDI".LS_XT_HDL_SW_UNLOCK := "SDI".LS_XT_HDL_SW_UNLOCK XOR "IDI".LS_XT_HDL_SW_UNLOCK;
       "PDI".LS_XT_HDL_SW_LOCK := "SDI".LS_XT_HDL_SW_LOCK XOR "IDI".LS_XT_HDL_SW_LOCK;
       "PDI".LS_GCH_DOOR_OP := "SDI".LS_GCH_DOOR_OP XOR "IDI".LS_GCH_DOOR_OP;
       "PDI".LS_GCH_DOOR_CL := "SDI".LS_GCH_DOOR_CL XOR "IDI".LS_GCH_DOOR_CL;
       "PDI".MCC_CONTACT_XT := "SDI".MCC_CONTACT_XT XOR "IDI".MCC_CONTACT_XT;
       "PDI".OIL_LVL_XT_SFT := "SDI".OIL_LVL_XT_SFT XOR "IDI".OIL_LVL_XT_SFT;
       "PDI".LS_XT_SFT_SRV_POS := "SDI".LS_XT_SFT_SRV_POS XOR "IDI".LS_XT_SFT_SRV_POS;
       "PDI".LS_XT_TOP_POS := "SDI".LS_XT_TOP_POS XOR "IDI".LS_XT_TOP_POS;
       "PDI".SLS_TCH_LFT := "SDI".SLS_TCH_LFT XOR "IDI".SLS_TCH_LFT;
       "PDI".XT_ROT_CAM_TRG := "SDI".XT_ROT_CAM_TRG XOR "IDI".XT_ROT_CAM_TRG;
       "PDI".MP_ENB_K8 := "SDI".MP_ENB_K8 XOR "IDI".MP_ENB_K8;
       "PDI".MP_ENB_K9 := "SDI".MP_ENB_K9 XOR "IDI".MP_ENB_K9;
       "PDI".LS_V3_OP := "SDI".LS_V3_OP XOR "IDI".LS_V3_OP;
       "PDI".LS_V3_CL := "SDI".LS_V3_CL XOR "IDI".LS_V3_CL;
       "PDI".FDR_LS_V3_2_OP := "SDI".FDR_LS_V3_2_OP XOR "IDI".FDR_LS_V3_2_OP;
       "PDI".FDR_LS_V3_2_CL := "SDI".FDR_LS_V3_2_CL XOR "IDI".FDR_LS_V3_2_CL;
       "PDI".LSR_SEN_OBJ_DET := "SDI".LSR_SEN_OBJ_DET XOR "IDI".LSR_SEN_OBJ_DET;
       "PDI".SPARE_280_5 := "SDI".SPARE_280_5 XOR "IDI".SPARE_280_5;
       "PDI".SPARE_280_6 := "SDI".SPARE_280_6 XOR "IDI".SPARE_280_6;
       "PDI".SPARE_280_7 := "SDI".SPARE_280_7 XOR "IDI".SPARE_280_7;
       "PDI".LS_V11_OP := "SDI".LS_V11_OP XOR "IDI".LS_V11_OP;
       "PDI".LS_V11_CL := "SDI".LS_V11_CL XOR "IDI".LS_V11_CL;
       "PDI".FDR_HOP_CON := "SDI".FDR_HOP_CON XOR "IDI".FDR_HOP_CON;
   ELSE

